LIN {X 0,Y 312.759,Z 483.247,A -85,B 0,C 180,E1 -15907.542,E2 -15907.542} C_VEL
LIN {X 0,Y 310.981,Z 494.774,A -85,B 0,C 180,E1 -15908.976,E2 -15908.976} C_VEL
LIN {X 0,Y 309.46,Z 504.322,A -85,B 0,C 180,E1 -15910.429,E2 -15910.429} C_VEL
LIN {X 0,Y 307.774,Z 514.927,A -85,B 0,C 180,E1 -15912.389,E2 -15912.389} C_VEL
LIN {X 0,Y 306.512,Z 523.604,A -85,B 0,C 180,E1 -15914.368,E2 -15914.368} C_VEL
LIN {X 0,Y 305.528,Z 530.802,A -85,B 0,C 180,E1 -15916.363,E2 -15916.363} C_VEL
LIN {X 0,Y 304.51,Z 537.588,A -85,B 0,C 180,E1 -15918.687,E2 -15918.687} C_VEL
LIN {X 0,Y 304.054,Z 542.26,A -85,B 0,C 180,E1 -15920.689,E2 -15920.689} C_VEL
LIN {X 0,Y 303.769,Z 545.92,A -85,B 0,C 180,E1 -15922.69,E2 -15922.69} C_VEL
LIN {X 0,Y 303.596,Z 548.706,A -85,B 0,C 180,E1 -15924.687,E2 -15924.687} C_VEL
LIN {X 0,Y 303.597,Z 551.095,A -85,B 0,C 180,E1 -15927.346,E2 -15927.346} C_VEL
LIN {X 0,Y 303.603,Z 552.04,A -85,B 0,C 180,E1 -15930,E2 -15930} C_VEL
LIN {X 0,Y 303.597,Z 551.554,A -85,B 0,C 180,E1 -15932.654,E2 -15932.654} C_VEL
LIN {X 0,Y 303.616,Z 549.633,A -85,B 0,C 180,E1 -15935.313,E2 -15935.313} C_VEL
LIN {X 0,Y 303.869,Z 546.198,A -85,B 0,C 180,E1 -15937.977,E2 -15937.977} C_VEL
LIN {X 0,Y 304.429,Z 541.183,A -85,B 0,C 180,E1 -15940.643,E2 -15940.643} C_VEL
LIN {X 0,Y 305.184,Z 536.305,A -85,B 0,C 180,E1 -15942.637,E2 -15942.637} C_VEL
LIN {X 0,Y 306.367,Z 529.293,A -85,B 0,C 180,E1 -15944.93,E2 -15944.93} C_VEL
LIN {X 0,Y 307.58,Z 521.737,A -85,B 0,C 180,E1 -15946.937,E2 -15946.937} C_VEL
LIN {X 0,Y 309.196,Z 512.715,A -85,B 0,C 180,E1 -15948.899,E2 -15948.899} C_VEL
LIN {X 0,Y 311.197,Z 501.739,A -85,B 0,C 180,E1 -15950.836,E2 -15950.836} C_VEL
LIN {X 0,Y 313.164,Z 490.536,A -85,B 0,C 180,E1 -15952.427,E2 -15952.427} C_VEL
LIN {X 0,Y 314.9,Z 478.707,A -85,B 0,C 180,E1 -15953.788,E2 -15953.788} C_VEL
LIN {X 0,Y 316.57,Z 465.924,A -85,B 0,C 180,E1 -15954.948,E2 -15954.948} C_VEL
LIN {X 0,Y 318.089,Z 452.516,A -85,B 0,C 180,E1 -15955.872,E2 -15955.872} C_VEL
LIN {X 0,Y 319.331,Z 438.667,A -85,B 0,C 180,E1 -15956.554,E2 -15956.554} C_VEL
LIN {X 0,Y 320.091,Z 424.187,A -85,B 0,C 180,E1 -15957.014,E2 -15957.014} C_VEL
LIN {X 0,Y 322.808,Z 332.95,A -85,B 0,C 180,E1 -15959.123,E2 -15959.123} C_VEL
LIN {X 0,Y 319.728,Z 313.724,A -85,B 0,C 180,E1 -15959.933,E2 -15959.933} C_VEL
LIN {X 0,Y 313.64,Z 300.106,A -85,B 0,C 180,E1 -15960.977,E2 -15960.977} C_VEL
LIN {X 0,Y 310.945,Z 288.941,A -85,B 0,C 180,E1 -15964.089,E2 -15964.089} C_VEL
LIN {X 0,Y 307.491,Z 276.823,A -85,B 0,C 180,E1 -15967.82,E2 -15967.82} C_VEL
LIN {X 0,Y 305.493,Z 270.13,A -85,B 0,C 180,E1 -15970.101,E2 -15970.101} C_VEL
LIN {X 0,Y 305.488,Z 270.046,A -85,B 0,C 180,E1 -15973.643,E2 -15973.643} C_VEL
LIN {X 0,Y 305.46,Z 270.051,A -85,B 0,C 180,E1 -15977.412,E2 -15977.412} C_VEL
LIN {X 0,Y 305.491,Z 270.058,A -85,B 0,C 180,E1 -15981.6,E2 -15981.6} C_VEL
LIN {X 0,Y 305.458,Z 270.04,A -85,B 0,C 180,E1 -15984.887,E2 -15984.887} C_VEL
LIN {X 0,Y 305.448,Z 270.049,A -85,B 0,C 180,E1 -15988.355,E2 -15988.355} C_VEL
LIN {X 0,Y 305.516,Z 270.026,A -85,B 0,C 180,E1 -15991.114,E2 -15991.114} C_VEL
LIN {X 0,Y 305.567,Z 270.047,A -85,B 0,C 180,E1 -15994.088,E2 -15994.088} C_VEL
LIN {X 0,Y 305.496,Z 270.052,A -85,B 0,C 180,E1 -15998.403,E2 -15998.403} C_VEL
LIN {X 0,Y 305.585,Z 270.044,A -85,B 0,C 180,E1 -16001.218,E2 -16001.218} C_VEL
LIN {X 0,Y 305.644,Z 270.035,A -85,B 0,C 180,E1 -16005.349,E2 -16005.349} C_VEL
LIN {X 0,Y 305.633,Z 270.033,A -85,B 0,C 180,E1 -16009.4,E2 -16009.4} C_VEL
LIN {X 0,Y 305.803,Z 270.006,A -85,B 0,C 180,E1 -16012.074,E2 -16012.074} C_VEL
LIN {X 0,Y 305.683,Z 270.032,A -85,B 0,C 180,E1 -16014.724,E2 -16014.724} C_VEL
LIN {X 0,Y 305.952,Z 269.994,A -85,B 0,C 180,E1 -16018.684,E2 -16018.684} C_VEL
LIN {X 0,Y 305.952,Z 269.991,A -85,B 0,C 180,E1 -16021.317,E2 -16021.317} C_VEL
LIN {X 0,Y 305.848,Z 270.002,A -85,B 0,C 180,E1 -16026.598,E2 -16026.598} C_VEL
LIN {X 0,Y 305.732,Z 270.028,A -85,B 0,C 180,E1 -16029.26,E2 -16029.26} C_VEL
LIN {X 0,Y 305.585,Z 270.044,A -85,B 0,C 180,E1 -16033.297,E2 -16033.297} C_VEL
LIN {X 0,Y 305.59,Z 270.034,A -85,B 0,C 180,E1 -16036.021,E2 -16036.021} C_VEL
LIN {X 0,Y 305.573,Z 270.038,A -85,B 0,C 180,E1 -16039.445,E2 -16039.445} C_VEL
LIN {X 0,Y 305.487,Z 270.053,A -85,B 0,C 180,E1 -16043.042,E2 -16043.042} C_VEL
LIN {X 0,Y 305.544,Z 270.05,A -85,B 0,C 180,E1 -16046.228,E2 -16046.228} C_VEL
LIN {X 0,Y 305.485,Z 270.027,A -85,B 0,C 180,E1 -16049.048,E2 -16049.048} C_VEL
LIN {X 0,Y 305.44,Z 270.064,A -85,B 0,C 180,E1 -16051.953,E2 -16051.953} C_VEL
LIN {X 0,Y 305.461,Z 270.037,A -85,B 0,C 180,E1 -16055.114,E2 -16055.114} C_VEL
LIN {X 0,Y 305.466,Z 270.052,A -85,B 0,C 180,E1 -16058.534,E2 -16058.534} C_VEL
LIN {X 0,Y 305.455,Z 270.06,A -85,B 0,C 180,E1 -16062.587,E2 -16062.587} C_VEL
LIN {X 0,Y 305.426,Z 270.063,A -85,B 0,C 180,E1 -16066.346,E2 -16066.346} C_VEL
LIN {X 0,Y 305.472,Z 270.249,A -85,B 0,C 180,E1 -16067.75,E2 -16067.75} C_VEL
LIN {X 0,Y 308.474,Z 280.592,A -85,B 0,C 180,E1 -16071.315,E2 -16071.315} C_VEL
LIN {X 0,Y 311.024,Z 290.406,A -85,B 0,C 180,E1 -16074.437,E2 -16074.437} C_VEL
LIN {X 0,Y 313.705,Z 302.514,A -85,B 0,C 180,E1 -16078.011,E2 -16078.011} C_VEL
LIN {X 0,Y 314.541,Z 307.647,A -85,B 0,C 180,E1 -16079.448,E2 -16079.448} C_VEL
LIN {X 0,Y 314.073,Z 310.802,A -85,B 0,C 180,E1 -16080.151,E2 -16080.151} C_VEL
LIN {X 0,Y 319.423,Z 338.198,A -85,B 0,C 180,E1 -16081.396,E2 -16081.396} C_VEL
LIN {X 0,Y 321.917,Z 352.925,A -85,B 0,C 180,E1 -16081.99,E2 -16081.99} C_VEL
LIN {X 0,Y 319.923,Z 427.545,A -85,B 0,C 180,E1 -16083.587,E2 -16083.587} C_VEL
LIN {X 0,Y 318.95,Z 440.96,A -85,B 0,C 180,E1 -16084.116,E2 -16084.116} C_VEL
LIN {X 0,Y 317.867,Z 453.812,A -85,B 0,C 180,E1 -16084.898,E2 -16084.898} C_VEL
LIN {X 0,Y 316.415,Z 466.19,A -85,B 0,C 180,E1 -16085.922,E2 -16085.922} C_VEL
LIN {X 0,Y 314.619,Z 477.746,A -85,B 0,C 180,E1 -16087.162,E2 -16087.162} C_VEL
LIN {X 0,Y 312.748,Z 488.241,A -85,B 0,C 180,E1 -16088.583,E2 -16088.583} C_VEL
LIN {X 0,Y 310.959,Z 497.743,A -85,B 0,C 180,E1 -16090.183,E2 -16090.183} C_VEL
LIN {X 0,Y 309.3,Z 505.574,A -85,B 0,C 180,E1 -16091.794,E2 -16091.794} C_VEL
LIN {X 0,Y 307.718,Z 513.396,A -85,B 0,C 180,E1 -16093.776,E2 -16093.776} C_VEL
LIN {X 0,Y 306.336,Z 520.446,A -85,B 0,C 180,E1 -16096.061,E2 -16096.061} C_VEL
LIN {X 0,Y 305.226,Z 525.27,A -85,B 0,C 180,E1 -16098.04,E2 -16098.04} C_VEL
LIN {X 0,Y 304.604,Z 529.037,A -85,B 0,C 180,E1 -16100.035,E2 -16100.035} C_VEL
LIN {X 0,Y 304.12,Z 531.847,A -85,B 0,C 180,E1 -16102.03,E2 -16102.03} C_VEL
LIN {X 0,Y 303.748,Z 534.172,A -85,B 0,C 180,E1 -16104.69,E2 -16104.69} C_VEL
LIN {X 0,Y 303.715,Z 534.785,A -85,B 0,C 180,E1 -16106.019,E2 -16106.019} C_VEL
LIN {X 0,Y 303.602,Z 534.951,A -85,B 0,C 180,E1 -16108.674,E2 -16108.674} C_VEL
LIN {X 0,Y 303.683,Z 533.622,A -85,B 0,C 180,E1 -16111.326,E2 -16111.326} C_VEL
LIN {X 0,Y 304.084,Z 530.811,A -85,B 0,C 180,E1 -16113.976,E2 -16113.976} C_VEL
LIN {X 0,Y 304.569,Z 527.648,A -85,B 0,C 180,E1 -16115.96,E2 -16115.96} C_VEL
LIN {X 0,Y 305.245,Z 523.152,A -85,B 0,C 180,E1 -16118.09,E2 -16118.09} C_VEL
LIN {X 0,Y 306.021,Z 518.261,A -85,B 0,C 180,E1 -16119.918,E2 -16119.918} C_VEL
LIN {X 0,Y 307.428,Z 510.543,A -85,B 0,C 180,E1 -16122.208,E2 -16122.208} C_VEL
LIN {X 0,Y 308.915,Z 502.223,A -85,B 0,C 180,E1 -16124.156,E2 -16124.156} C_VEL
LIN {X 0,Y 310.409,Z 493.744,A -85,B 0,C 180,E1 -16125.765,E2 -16125.765} C_VEL
LIN {X 0,Y 312.086,Z 483.367,A -85,B 0,C 180,E1 -16127.36,E2 -16127.36} C_VEL
LIN {X 0,Y 313.701,Z 471.745,A -85,B 0,C 180,E1 -16128.787,E2 -16128.787} C_VEL
LIN {X 0,Y 315.026,Z 462.036,A -85,B 0,C 180,E1 -16129.72,E2 -16129.72} C_VEL
LIN {X 0,Y 316.343,Z 449.727,A -85,B 0,C 180,E1 -16130.651,E2 -16130.651} C_VEL
LIN {X 0,Y 317.274,Z 436.502,A -85,B 0,C 180,E1 -16131.368,E2 -16131.368} C_VEL
LIN {X 0,Y 317.974,Z 423.135,A -85,B 0,C 180,E1 -16131.816,E2 -16131.816} C_VEL
LIN {X 0,Y 319.599,Z 351.308,A -85,B 0,C 180,E1 -16133.344,E2 -16133.344} C_VEL
LIN {X 0,Y 314.658,Z 321.72,A -85,B 0,C 180,E1 -16134.479,E2 -16134.479} C_VEL
LIN {X 0,Y 312.643,Z 310.757,A -85,B 0,C 180,E1 -16134.972,E2 -16134.972} C_VEL
LIN {X 0,Y 313.465,Z 303.711,A -85,B 0,C 180,E1 -16136.641,E2 -16136.641} C_VEL
LIN {X 0,Y 311.277,Z 292.524,A -85,B 0,C 180,E1 -16139.782,E2 -16139.782} C_VEL
LIN {X 0,Y 308.2,Z 280.123,A -85,B 0,C 180,E1 -16143.526,E2 -16143.526} C_VEL
LIN {X 0,Y 305.574,Z 270.458,A -85,B 0,C 180,E1 -16146.661,E2 -16146.661} C_VEL
LIN {X 0,Y 305.318,Z 270.1,A -85,B 0,C 180,E1 -16146.986,E2 -16146.986} C_VEL
LIN {X 0,Y 302.785,Z 270.39,A -85,B 0,C 180,E1 -16148.741,E2 -16148.741} C_VEL
LIN {X 0,Y 299.323,Z 271.015,A -85,B 0,C 180,E1 -16150.95,E2 -16150.95} C_VEL
LIN {X 0,Y 298.422,Z 270.949,A -85,B 0,C 180,E1 -16152.109,E2 -16152.109} C_VEL
LIN {X 0,Y 298.364,Z 270.938,A -85,B 0,C 180,E1 -16152.501,E2 -16152.501} C_VEL
LIN {X 0,Y 298.402,Z 270.937,A -85,B 0,C 180,E1 -16156.92,E2 -16156.92} C_VEL
LIN {X 0,Y 298.413,Z 270.917,A -85,B 0,C 180,E1 -16161.003,E2 -16161.003} C_VEL
LIN {X 0,Y 298.43,Z 270.933,A -85,B 0,C 180,E1 -16163.931,E2 -16163.931} C_VEL
LIN {X 0,Y 298.393,Z 270.924,A -85,B 0,C 180,E1 -16167.982,E2 -16167.982} C_VEL
LIN {X 0,Y 298.467,Z 270.922,A -85,B 0,C 180,E1 -16171.904,E2 -16171.904} C_VEL
LIN {X 0,Y 298.482,Z 270.923,A -85,B 0,C 180,E1 -16174.923,E2 -16174.923} C_VEL
LIN {X 0,Y 298.446,Z 270.927,A -85,B 0,C 180,E1 -16179.314,E2 -16179.314} C_VEL
LIN {X 0,Y 298.534,Z 270.922,A -85,B 0,C 180,E1 -16182.179,E2 -16182.179} C_VEL
LIN {X 0,Y 298.589,Z 270.905,A -85,B 0,C 180,E1 -16184.994,E2 -16184.994} C_VEL
LIN {X 0,Y 298.587,Z 270.908,A -85,B 0,C 180,E1 -16189.146,E2 -16189.146} C_VEL
LIN {X 0,Y 298.736,Z 270.895,A -85,B 0,C 180,E1 -16191.885,E2 -16191.885} C_VEL
LIN {X 0,Y 298.652,Z 270.897,A -85,B 0,C 180,E1 -16194.598,E2 -16194.598} C_VEL
LIN {X 0,Y 298.918,Z 270.874,A -85,B 0,C 180,E1 -16198.652,E2 -16198.652} C_VEL
LIN {X 0,Y 298.918,Z 270.865,A -85,B 0,C 180,E1 -16201.347,E2 -16201.347} C_VEL
LIN {X 0,Y 298.792,Z 270.881,A -85,B 0,C 180,E1 -16206.754,E2 -16206.754} C_VEL
LIN {X 0,Y 298.675,Z 270.903,A -85,B 0,C 180,E1 -16209.48,E2 -16209.48} C_VEL
LIN {X 0,Y 298.546,Z 270.922,A -85,B 0,C 180,E1 -16213.615,E2 -16213.615} C_VEL
LIN {X 0,Y 298.543,Z 270.912,A -85,B 0,C 180,E1 -16216.409,E2 -16216.409} C_VEL
LIN {X 0,Y 298.506,Z 270.921,A -85,B 0,C 180,E1 -16219.655,E2 -16219.655} C_VEL
LIN {X 0,Y 298.452,Z 270.932,A -85,B 0,C 180,E1 -16223.598,E2 -16223.598} C_VEL
LIN {X 0,Y 298.485,Z 270.93,A -85,B 0,C 180,E1 -16226.574,E2 -16226.574} C_VEL
LIN {X 0,Y 298.416,Z 270.908,A -85,B 0,C 180,E1 -16229.641,E2 -16229.641} C_VEL
LIN {X 0,Y 298.391,Z 270.936,A -85,B 0,C 180,E1 -16232.8,E2 -16232.8} C_VEL
LIN {X 0,Y 298.442,Z 270.909,A -85,B 0,C 180,E1 -16236.808,E2 -16236.808} C_VEL
LIN {X 0,Y 298.383,Z 270.93,A -85,B 0,C 180,E1 -16241.088,E2 -16241.088} C_VEL
LIN {X 0,Y 298.385,Z 270.935,A -85,B 0,C 180,E1 -16245.042,E2 -16245.042} C_VEL
LIN {X 0,Y 298.384,Z 270.886,A -85,B 0,C 180,E1 -16248.913,E2 -16248.913} C_VEL
LIN {X 0,Y 298.422,Z 271.119,A -85,B 0,C 180,E1 -16250.769,E2 -16250.769} C_VEL
LIN {X 0,Y 301.752,Z 282.523,A -85,B 0,C 180,E1 -16254.391,E2 -16254.391} C_VEL
LIN {X 0,Y 304.525,Z 293.397,A -85,B 0,C 180,E1 -16257.58,E2 -16257.58} C_VEL
LIN {X 0,Y 306.122,Z 300.383,A -85,B 0,C 180,E1 -16259.437,E2 -16259.437} C_VEL
LIN {X 0,Y 311.319,Z 312.764,A -85,B 0,C 180,E1 -16260.308,E2 -16260.308} C_VEL
LIN {X 0,Y 314.225,Z 333.621,A -85,B 0,C 180,E1 -16261.127,E2 -16261.127} C_VEL
LIN {X 0,Y 311.299,Z 430.528,A -85,B 0,C 180,E1 -16263.43,E2 -16263.43} C_VEL
LIN {X 0,Y 310.325,Z 445.033,A -85,B 0,C 180,E1 -16264.019,E2 -16264.019} C_VEL
LIN {X 0,Y 309.172,Z 457.738,A -85,B 0,C 180,E1 -16264.773,E2 -16264.773} C_VEL
LIN {X 0,Y 307.655,Z 471.105,A -85,B 0,C 180,E1 -16265.838,E2 -16265.838} C_VEL
LIN {X 0,Y 306.161,Z 482.751,A -85,B 0,C 180,E1 -16267.031,E2 -16267.031} C_VEL
LIN {X 0,Y 304.322,Z 494.343,A -85,B 0,C 180,E1 -16268.493,E2 -16268.493} C_VEL
LIN {X 0,Y 302.685,Z 503.937,A -85,B 0,C 180,E1 -16269.973,E2 -16269.973} C_VEL
LIN {X 0,Y 300.971,Z 514.584,A -85,B 0,C 180,E1 -16271.977,E2 -16271.977} C_VEL
LIN {X 0,Y 299.496,Z 523.967,A -85,B 0,C 180,E1 -16274.176,E2 -16274.176} C_VEL
LIN {X 0,Y 298.548,Z 530.514,A -85,B 0,C 180,E1 -16276.038,E2 -16276.038} C_VEL
LIN {X 0,Y 297.511,Z 537.328,A -85,B 0,C 180,E1 -16278.417,E2 -16278.417} C_VEL
LIN {X 0,Y 297.004,Z 542.007,A -85,B 0,C 180,E1 -16280.466,E2 -16280.466} C_VEL
LIN {X 0,Y 296.69,Z 545.683,A -85,B 0,C 180,E1 -16282.514,E2 -16282.514} C_VEL
LIN {X 0,Y 296.511,Z 548.482,A -85,B 0,C 180,E1 -16284.56,E2 -16284.56} C_VEL
LIN {X 0,Y 296.522,Z 550.884,A -85,B 0,C 180,E1 -16287.283,E2 -16287.283} C_VEL
LIN {X 0,Y 296.518,Z 551.839,A -85,B 0,C 180,E1 -16290,E2 -16290} C_VEL
LIN {X 0,Y 296.522,Z 551.362,A -85,B 0,C 180,E1 -16292.717,E2 -16292.717} C_VEL
LIN {X 0,Y 296.545,Z 549.383,A -85,B 0,C 180,E1 -16295.509,E2 -16295.509} C_VEL
LIN {X 0,Y 296.814,Z 546.027,A -85,B 0,C 180,E1 -16298.168,E2 -16298.168} C_VEL
LIN {X 0,Y 297.388,Z 541.019,A -85,B 0,C 180,E1 -16300.898,E2 -16300.898} C_VEL
LIN {X 0,Y 298.229,Z 536.149,A -85,B 0,C 180,E1 -16302.937,E2 -16302.937} C_VEL
LIN {X 0,Y 299.259,Z 530.192,A -85,B 0,C 180,E1 -16304.971,E2 -16304.971} C_VEL
LIN {X 0,Y 300.527,Z 522.967,A -85,B 0,C 180,E1 -16306.997,E2 -16306.997} C_VEL
LIN {X 0,Y 302.149,Z 514.222,A -85,B 0,C 180,E1 -16309.004,E2 -16309.004} C_VEL
LIN {X 0,Y 304.15,Z 503.571,A -85,B 0,C 180,E1 -16310.987,E2 -16310.987} C_VEL
LIN {X 0,Y 306.156,Z 492.777,A -85,B 0,C 180,E1 -16312.613,E2 -16312.613} C_VEL
LIN {X 0,Y 308.1,Z 480.527,A -85,B 0,C 180,E1 -16314.112,E2 -16314.112} C_VEL
LIN {X 0,Y 309.917,Z 467.747,A -85,B 0,C 180,E1 -16315.342,E2 -16315.342} C_VEL
LIN {X 0,Y 311.443,Z 454.922,A -85,B 0,C 180,E1 -16316.286,E2 -16316.286} C_VEL
LIN {X 0,Y 312.757,Z 441.147,A -85,B 0,C 180,E1 -16317.022,E2 -16317.022} C_VEL
LIN {X 0,Y 313.656,Z 426.797,A -85,B 0,C 180,E1 -16317.525,E2 -16317.525} C_VEL
LIN {X 0,Y 316.583,Z 334.1,A -85,B 0,C 180,E1 -16319.709,E2 -16319.709} C_VEL
LIN {X 0,Y 313.725,Z 316.254,A -85,B 0,C 180,E1 -16320.485,E2 -16320.485} C_VEL
LIN {X 0,Y 306.546,Z 300.388,A -85,B 0,C 180,E1 -16321.739,E2 -16321.739} C_VEL
LIN {X 0,Y 303.827,Z 289.344,A -85,B 0,C 180,E1 -16324.924,E2 -16324.924} C_VEL
LIN {X 0,Y 300.648,Z 278.286,A -85,B 0,C 180,E1 -16328.456,E2 -16328.456} C_VEL
LIN {X 0,Y 298.452,Z 271.029,A -85,B 0,C 180,E1 -16330.983,E2 -16330.983} C_VEL
LIN {X 0,Y 298.456,Z 270.928,A -85,B 0,C 180,E1 -16333.115,E2 -16333.115} C_VEL
LIN {X 0,Y 298.429,Z 270.935,A -85,B 0,C 180,E1 -16336.926,E2 -16336.926} C_VEL
LIN {X 0,Y 298.411,Z 270.94,A -85,B 0,C 180,E1 -16341.003,E2 -16341.003} C_VEL
LIN {X 0,Y 298.416,Z 270.912,A -85,B 0,C 180,E1 -16343.93,E2 -16343.93} C_VEL
LIN {X 0,Y 298.391,Z 270.933,A -85,B 0,C 180,E1 -16347.983,E2 -16347.983} C_VEL
LIN {X 0,Y 298.459,Z 270.915,A -85,B 0,C 180,E1 -16351.904,E2 -16351.904} C_VEL
LIN {X 0,Y 298.481,Z 270.924,A -85,B 0,C 180,E1 -16354.924,E2 -16354.924} C_VEL
LIN {X 0,Y 298.445,Z 270.925,A -85,B 0,C 180,E1 -16359.315,E2 -16359.315} C_VEL
LIN {X 0,Y 298.533,Z 270.921,A -85,B 0,C 180,E1 -16362.179,E2 -16362.179} C_VEL
LIN {X 0,Y 298.589,Z 270.912,A -85,B 0,C 180,E1 -16364.995,E2 -16364.995} C_VEL
LIN {X 0,Y 298.588,Z 270.909,A -85,B 0,C 180,E1 -16369.147,E2 -16369.147} C_VEL
LIN {X 0,Y 298.75,Z 270.886,A -85,B 0,C 180,E1 -16371.886,E2 -16371.886} C_VEL
LIN {X 0,Y 298.654,Z 270.907,A -85,B 0,C 180,E1 -16374.599,E2 -16374.599} C_VEL
LIN {X 0,Y 298.919,Z 270.87,A -85,B 0,C 180,E1 -16378.653,E2 -16378.653} C_VEL
LIN {X 0,Y 298.919,Z 270.867,A -85,B 0,C 180,E1 -16381.348,E2 -16381.348} C_VEL
LIN {X 0,Y 298.793,Z 270.879,A -85,B 0,C 180,E1 -16386.754,E2 -16386.754} C_VEL
LIN {X 0,Y 298.677,Z 270.906,A -85,B 0,C 180,E1 -16389.481,E2 -16389.481} C_VEL
LIN {X 0,Y 298.548,Z 270.922,A -85,B 0,C 180,E1 -16393.616,E2 -16393.616} C_VEL
LIN {X 0,Y 298.545,Z 270.913,A -85,B 0,C 180,E1 -16396.409,E2 -16396.409} C_VEL
LIN {X 0,Y 298.508,Z 270.917,A -85,B 0,C 180,E1 -16399.655,E2 -16399.655} C_VEL
LIN {X 0,Y 298.455,Z 270.925,A -85,B 0,C 180,E1 -16403.599,E2 -16403.599} C_VEL
LIN {X 0,Y 298.487,Z 270.925,A -85,B 0,C 180,E1 -16406.575,E2 -16406.575} C_VEL
LIN {X 0,Y 298.414,Z 270.909,A -85,B 0,C 180,E1 -16409.642,E2 -16409.642} C_VEL
LIN {X 0,Y 298.393,Z 270.939,A -85,B 0,C 180,E1 -16412.801,E2 -16412.801} C_VEL
LIN {X 0,Y 298.463,Z 270.925,A -85,B 0,C 180,E1 -16416.813,E2 -16416.813} C_VEL
LIN {X 0,Y 298.386,Z 270.928,A -85,B 0,C 180,E1 -16421.088,E2 -16421.088} C_VEL
LIN {X 0,Y 298.399,Z 270.931,A -85,B 0,C 180,E1 -16423.104,E2 -16423.104} C_VEL
LIN {X 0,Y 298.422,Z 271.135,A -85,B 0,C 180,E1 -16426.847,E2 -16426.847} C_VEL
LIN {X 0,Y 301.273,Z 280.862,A -85,B 0,C 180,E1 -16430.338,E2 -16430.338} C_VEL
LIN {X 0,Y 304.224,Z 291.819,A -85,B 0,C 180,E1 -16433.955,E2 -16433.955} C_VEL
LIN {X 0,Y 307.023,Z 304.814,A -85,B 0,C 180,E1 -16437.884,E2 -16437.884} C_VEL
LIN {X 0,Y 307.738,Z 309.703,A -85,B 0,C 180,E1 -16439.271,E2 -16439.271} C_VEL
LIN {X 0,Y 307.638,Z 310.773,A -85,B 0,C 180,E1 -16439.46,E2 -16439.46} C_VEL
LIN {X 0,Y 312.585,Z 335.948,A -85,B 0,C 180,E1 -16440.646,E2 -16440.646} C_VEL
LIN {X 0,Y 315.647,Z 354.231,A -85,B 0,C 180,E1 -16441.408,E2 -16441.408} C_VEL
LIN {X 0,Y 313.648,Z 426.468,A -85,B 0,C 180,E1 -16442.971,E2 -16442.971} C_VEL
LIN {X 0,Y 312.739,Z 439.521,A -85,B 0,C 180,E1 -16443.472,E2 -16443.472} C_VEL
LIN {X 0,Y 311.534,Z 452.773,A -85,B 0,C 180,E1 -16444.262,E2 -16444.262} C_VEL
LIN {X 0,Y 310.122,Z 464.797,A -85,B 0,C 180,E1 -16445.245,E2 -16445.245} C_VEL
LIN {X 0,Y 308.33,Z 476.561,A -85,B 0,C 180,E1 -16446.492,E2 -16446.492} C_VEL
LIN {X 0,Y 306.35,Z 487.287,A -85,B 0,C 180,E1 -16447.935,E2 -16447.935} C_VEL
LIN {X 0,Y 304.601,Z 496.096,A -85,B 0,C 180,E1 -16449.399,E2 -16449.399} C_VEL
LIN {X 0,Y 302.531,Z 505.695,A -85,B 0,C 180,E1 -16451.372,E2 -16451.372} C_VEL
LIN {X 0,Y 300.992,Z 512.839,A -85,B 0,C 180,E1 -16453.204,E2 -16453.204} C_VEL
LIN {X 0,Y 299.858,Z 518.72,A -85,B 0,C 180,E1 -16455.06,E2 -16455.06} C_VEL
LIN {X 0,Y 298.593,Z 523.933,A -85,B 0,C 180,E1 -16457.079,E2 -16457.079} C_VEL
LIN {X 0,Y 297.769,Z 528.04,A -85,B 0,C 180,E1 -16459.116,E2 -16459.116} C_VEL
LIN {X 0,Y 297.412,Z 530.234,A -85,B 0,C 180,E1 -16460.479,E2 -16460.479} C_VEL
LIN {X 0,Y 297.07,Z 532.019,A -85,B 0,C 180,E1 -16461.84,E2 -16461.84} C_VEL
LIN {X 0,Y 296.672,Z 534.356,A -85,B 0,C 180,E1 -16464.563,E2 -16464.563} C_VEL
LIN {X 0,Y 296.574,Z 535.24,A -85,B 0,C 180,E1 -16467.283,E2 -16467.283} C_VEL
LIN {X 0,Y 296.528,Z 534.688,A -85,B 0,C 180,E1 -16470,E2 -16470} C_VEL
LIN {X 0,Y 296.762,Z 532.631,A -85,B 0,C 180,E1 -16472.715,E2 -16472.715} C_VEL
LIN {X 0,Y 297.355,Z 529.071,A -85,B 0,C 180,E1 -16475.425,E2 -16475.425} C_VEL
LIN {X 0,Y 297.897,Z 525.39,A -85,B 0,C 180,E1 -16477.398,E2 -16477.398} C_VEL
LIN {X 0,Y 298.696,Z 520.427,A -85,B 0,C 180,E1 -16479.48,E2 -16479.48} C_VEL
LIN {X 0,Y 299.801,Z 514.388,A -85,B 0,C 180,E1 -16481.493,E2 -16481.493} C_VEL
LIN {X 0,Y 301.287,Z 506.941,A -85,B 0,C 180,E1 -16483.489,E2 -16483.489} C_VEL
LIN {X 0,Y 302.676,Z 499.386,A -85,B 0,C 180,E1 -16485.142,E2 -16485.142} C_VEL
LIN {X 0,Y 304.386,Z 489.266,A -85,B 0,C 180,E1 -16486.947,E2 -16486.947} C_VEL
LIN {X 0,Y 306.108,Z 479.014,A -85,B 0,C 180,E1 -16488.402,E2 -16488.402} C_VEL
LIN {X 0,Y 307.518,Z 469.278,A -85,B 0,C 180,E1 -16489.526,E2 -16489.526} C_VEL
LIN {X 0,Y 309.054,Z 457.012,A -85,B 0,C 180,E1 -16490.638,E2 -16490.638} C_VEL
LIN {X 0,Y 310.233,Z 444.565,A -85,B 0,C 180,E1 -16491.486,E2 -16491.486} C_VEL
LIN {X 0,Y 311.151,Z 431.625,A -85,B 0,C 180,E1 -16492.09,E2 -16492.09} C_VEL
LIN {X 0,Y 311.7,Z 416.204,A -85,B 0,C 180,E1 -16492.508,E2 -16492.508} C_VEL
LIN {X 0,Y 313.152,Z 351.889,A -85,B 0,C 180,E1 -16493.901,E2 -16493.901} C_VEL
LIN {X 0,Y 308.103,Z 321.447,A -85,B 0,C 180,E1 -16495.108,E2 -16495.108} C_VEL
LIN {X 0,Y 306.091,Z 310.752,A -85,B 0,C 180,E1 -16495.599,E2 -16495.599} C_VEL
LIN {X 0,Y 306.673,Z 305.551,A -85,B 0,C 180,E1 -16496.829,E2 -16496.829} C_VEL
LIN {X 0,Y 304.742,Z 295.455,A -85,B 0,C 180,E1 -16499.723,E2 -16499.723} C_VEL
LIN {X 0,Y 301.852,Z 283.472,A -85,B 0,C 180,E1 -16503.4,E2 -16503.4} C_VEL
LIN {X 0,Y 298.928,Z 272.785,A -85,B 0,C 180,E1 -16506.93,E2 -16506.93} C_VEL
LIN {X 0,Y 298.458,Z 270.999,A -85,B 0,C 180,E1 -16507.618,E2 -16507.618} C_VEL
LIN {X 0,Y 298.384,Z 270.929,A -85,B 0,C 180,E1 -16511.261,E2 -16511.261} C_VEL
LIN {X 0,Y 298.364,Z 270.938,A -85,B 0,C 180,E1 -16512.501,E2 -16512.501} C_VEL
LIN {X 0,Y 297.738,Z 271.029,A -85,B 0,C 180,E1 -16513.628,E2 -16513.628} C_VEL
LIN {X 0,Y 294.904,Z 271.392,A -85,B 0,C 180,E1 -16515.463,E2 -16515.463} C_VEL
LIN {X 0,Y 292.47,Z 271.689,A -85,B 0,C 180,E1 -16516.953,E2 -16516.953} C_VEL
LIN {X 0,Y 291.413,Z 271.808,A -85,B 0,C 180,E1 -16518.106,E2 -16518.106} C_VEL
LIN {X 0,Y 291.322,Z 271.811,A -85,B 0,C 180,E1 -16518.498,E2 -16518.498} C_VEL
LIN {X 0,Y 291.363,Z 271.796,A -85,B 0,C 180,E1 -16521.159,E2 -16521.159} C_VEL
LIN {X 0,Y 291.383,Z 271.797,A -85,B 0,C 180,E1 -16524.628,E2 -16524.628} C_VEL
LIN {X 0,Y 291.37,Z 271.797,A -85,B 0,C 180,E1 -16527.95,E2 -16527.95} C_VEL
LIN {X 0,Y 291.382,Z 271.807,A -85,B 0,C 180,E1 -16531.158,E2 -16531.158} C_VEL
LIN {X 0,Y 291.418,Z 271.81,A -85,B 0,C 180,E1 -16534.271,E2 -16534.271} C_VEL
LIN {X 0,Y 291.377,Z 271.814,A -85,B 0,C 180,E1 -16537.299,E2 -16537.299} C_VEL
LIN {X 0,Y 291.455,Z 271.794,A -85,B 0,C 180,E1 -16540.269,E2 -16540.269} C_VEL
LIN {X 0,Y 291.536,Z 271.784,A -85,B 0,C 180,E1 -16544.634,E2 -16544.634} C_VEL
LIN {X 0,Y 291.531,Z 271.788,A -85,B 0,C 180,E1 -16548.88,E2 -16548.88} C_VEL
LIN {X 0,Y 291.683,Z 271.773,A -85,B 0,C 180,E1 -16551.687,E2 -16551.687} C_VEL
LIN {X 0,Y 291.622,Z 271.773,A -85,B 0,C 180,E1 -16554.468,E2 -16554.468} C_VEL
LIN {X 0,Y 291.884,Z 271.75,A -85,B 0,C 180,E1 -16558.62,E2 -16558.62} C_VEL
LIN {X 0,Y 291.884,Z 271.741,A -85,B 0,C 180,E1 -16561.379,E2 -16561.379} C_VEL
LIN {X 0,Y 291.741,Z 271.761,A -85,B 0,C 180,E1 -16566.918,E2 -16566.918} C_VEL
LIN {X 0,Y 291.624,Z 271.78,A -85,B 0,C 180,E1 -16569.712,E2 -16569.712} C_VEL
LIN {X 0,Y 291.516,Z 271.799,A -85,B 0,C 180,E1 -16573.95,E2 -16573.95} C_VEL
LIN {X 0,Y 291.482,Z 271.795,A -85,B 0,C 180,E1 -16576.818,E2 -16576.818} C_VEL
LIN {X 0,Y 291.446,Z 271.798,A -85,B 0,C 180,E1 -16579.875,E2 -16579.875} C_VEL
LIN {X 0,Y 291.395,Z 271.805,A -85,B 0,C 180,E1 -16584.205,E2 -16584.205} C_VEL
LIN {X 0,Y 291.418,Z 271.81,A -85,B 0,C 180,E1 -16587.272,E2 -16587.272} C_VEL
LIN {X 0,Y 291.332,Z 271.787,A -85,B 0,C 180,E1 -16590.437,E2 -16590.437} C_VEL
LIN {X 0,Y 291.34,Z 271.822,A -85,B 0,C 180,E1 -16593.699,E2 -16593.699} C_VEL
LIN {X 0,Y 291.372,Z 271.791,A -85,B 0,C 180,E1 -16597.254,E2 -16597.254} C_VEL
LIN {X 0,Y 291.329,Z 271.815,A -85,B 0,C 180,E1 -16600.643,E2 -16600.643} C_VEL
LIN {X 0,Y 291.312,Z 271.824,A -85,B 0,C 180,E1 -16604.397,E2 -16604.397} C_VEL
LIN {X 0,Y 291.323,Z 271.761,A -85,B 0,C 180,E1 -16608.405,E2 -16608.405} C_VEL
LIN {X 0,Y 291.356,Z 272,A -85,B 0,C 180,E1 -16609.918,E2 -16609.918} C_VEL
LIN {X 0,Y 294.772,Z 283.523,A -85,B 0,C 180,E1 -16613.724,E2 -16613.724} C_VEL
LIN {X 0,Y 297.888,Z 295.768,A -85,B 0,C 180,E1 -16617.42,E2 -16617.42} C_VEL
LIN {X 0,Y 298.984,Z 300.489,A -85,B 0,C 180,E1 -16618.698,E2 -16618.698} C_VEL
LIN {X 0,Y 305.18,Z 314.984,A -85,B 0,C 180,E1 -16619.767,E2 -16619.767} C_VEL
LIN {X 0,Y 307.879,Z 334.862,A -85,B 0,C 180,E1 -16620.566,E2 -16620.566} C_VEL
LIN {X 0,Y 304.805,Z 431.437,A -85,B 0,C 180,E1 -16622.911,E2 -16622.911} C_VEL
LIN {X 0,Y 303.785,Z 445.606,A -85,B 0,C 180,E1 -16623.509,E2 -16623.509} C_VEL
LIN {X 0,Y 302.616,Z 458.149,A -85,B 0,C 180,E1 -16624.279,E2 -16624.279} C_VEL
LIN {X 0,Y 301.108,Z 470.821,A -85,B 0,C 180,E1 -16625.309,E2 -16625.309} C_VEL
LIN {X 0,Y 299.594,Z 482.256,A -85,B 0,C 180,E1 -16626.498,E2 -16626.498} C_VEL
LIN {X 0,Y 297.684,Z 493.913,A -85,B 0,C 180,E1 -16627.989,E2 -16627.989} C_VEL
LIN {X 0,Y 295.968,Z 503.554,A -85,B 0,C 180,E1 -16629.498,E2 -16629.498} C_VEL
LIN {X 0,Y 294.161,Z 514.238,A -85,B 0,C 180,E1 -16631.545,E2 -16631.545} C_VEL
LIN {X 0,Y 292.656,Z 523.497,A -85,B 0,C 180,E1 -16633.749,E2 -16633.749} C_VEL
LIN {X 0,Y 291.585,Z 530.224,A -85,B 0,C 180,E1 -16635.697,E2 -16635.697} C_VEL
LIN {X 0,Y 290.527,Z 537.068,A -85,B 0,C 180,E1 -16638.135,E2 -16638.135} C_VEL
LIN {X 0,Y 289.971,Z 541.754,A -85,B 0,C 180,E1 -16640.232,E2 -16640.232} C_VEL
LIN {X 0,Y 289.638,Z 545.446,A -85,B 0,C 180,E1 -16642.331,E2 -16642.331} C_VEL
LIN {X 0,Y 289.409,Z 548.496,A -85,B 0,C 180,E1 -16644.648,E2 -16644.648} C_VEL
LIN {X 0,Y 289.425,Z 550.672,A -85,B 0,C 180,E1 -16647.216,E2 -16647.216} C_VEL
LIN {X 0,Y 289.435,Z 551.638,A -85,B 0,C 180,E1 -16650,E2 -16650} C_VEL
LIN {X 0,Y 289.425,Z 551.171,A -85,B 0,C 180,E1 -16652.784,E2 -16652.784} C_VEL
LIN {X 0,Y 289.475,Z 549.271,A -85,B 0,C 180,E1 -16655.573,E2 -16655.573} C_VEL
LIN {X 0,Y 289.751,Z 545.856,A -85,B 0,C 180,E1 -16658.368,E2 -16658.368} C_VEL
LIN {X 0,Y 290.357,Z 540.855,A -85,B 0,C 180,E1 -16661.165,E2 -16661.165} C_VEL
LIN {X 0,Y 291.256,Z 535.992,A -85,B 0,C 180,E1 -16663.252,E2 -16663.252} C_VEL
LIN {X 0,Y 292.59,Z 528.937,A -85,B 0,C 180,E1 -16665.667,E2 -16665.667} C_VEL
LIN {X 0,Y 294.19,Z 520.07,A -85,B 0,C 180,E1 -16668.093,E2 -16668.093} C_VEL
LIN {X 0,Y 296.074,Z 510.785,A -85,B 0,C 180,E1 -16670.132,E2 -16670.132} C_VEL
LIN {X 0,Y 298.083,Z 500.452,A -85,B 0,C 180,E1 -16671.98,E2 -16671.98} C_VEL
LIN {X 0,Y 300.042,Z 490.259,A -85,B 0,C 180,E1 -16673.465,E2 -16673.465} C_VEL
LIN {X 0,Y 302.026,Z 477.761,A -85,B 0,C 180,E1 -16674.945,E2 -16674.945} C_VEL
LIN {X 0,Y 303.726,Z 465.615,A -85,B 0,C 180,E1 -16676.081,E2 -16676.081} C_VEL
LIN {X 0,Y 305.387,Z 452.166,A -85,B 0,C 180,E1 -16677.033,E2 -16677.033} C_VEL
LIN {X 0,Y 306.707,Z 438.23,A -85,B 0,C 180,E1 -16677.739,E2 -16677.739} C_VEL
LIN {X 0,Y 307.45,Z 425.02,A -85,B 0,C 180,E1 -16678.175,E2 -16678.175} C_VEL
LIN {X 0,Y 310.352,Z 335.004,A -85,B 0,C 180,E1 -16680.331,E2 -16680.331} C_VEL
LIN {X 0,Y 307.879,Z 319.036,A -85,B 0,C 180,E1 -16681.037,E2 -16681.037} C_VEL
LIN {X 0,Y 299.844,Z 301.564,A -85,B 0,C 180,E1 -16682.457,E2 -16682.457} C_VEL
LIN {X 0,Y 299.313,Z 300.205,A -85,B 0,C 180,E1 -16682.638,E2 -16682.638} C_VEL
LIN {X 0,Y 296.675,Z 289.723,A -85,B 0,C 180,E1 -16685.82,E2 -16685.82} C_VEL
LIN {X 0,Y 293.625,Z 279.083,A -85,B 0,C 180,E1 -16689.354,E2 -16689.354} C_VEL
LIN {X 0,Y 291.404,Z 271.883,A -85,B 0,C 180,E1 -16691.983,E2 -16691.983} C_VEL
LIN {X 0,Y 291.345,Z 271.82,A -85,B 0,C 180,E1 -16696.358,E2 -16696.358} C_VEL
LIN {X 0,Y 291.383,Z 271.809,A -85,B 0,C 180,E1 -16700.517,E2 -16700.517} C_VEL
LIN {X 0,Y 291.41,Z 271.79,A -85,B 0,C 180,E1 -16702.92,E2 -16702.92} C_VEL
LIN {X 0,Y 291.341,Z 271.816,A -85,B 0,C 180,E1 -16706.301,E2 -16706.301} C_VEL
LIN {X 0,Y 291.383,Z 271.78,A -85,B 0,C 180,E1 -16710.26,E2 -16710.26} C_VEL
LIN {X 0,Y 291.413,Z 271.808,A -85,B 0,C 180,E1 -16714.272,E2 -16714.272} C_VEL
LIN {X 0,Y 291.377,Z 271.815,A -85,B 0,C 180,E1 -16717.3,E2 -16717.3} C_VEL
LIN {X 0,Y 291.454,Z 271.798,A -85,B 0,C 180,E1 -16720.27,E2 -16720.27} C_VEL
LIN {X 0,Y 291.551,Z 271.786,A -85,B 0,C 180,E1 -16724.624,E2 -16724.624} C_VEL
LIN {X 0,Y 291.532,Z 271.786,A -85,B 0,C 180,E1 -16728.881,E2 -16728.881} C_VEL
LIN {X 0,Y 291.701,Z 271.766,A -85,B 0,C 180,E1 -16731.689,E2 -16731.689} C_VEL
LIN {X 0,Y 291.624,Z 271.783,A -85,B 0,C 180,E1 -16734.469,E2 -16734.469} C_VEL
LIN {X 0,Y 291.885,Z 271.746,A -85,B 0,C 180,E1 -16738.621,E2 -16738.621} C_VEL
LIN {X 0,Y 291.885,Z 271.742,A -85,B 0,C 180,E1 -16741.38,E2 -16741.38} C_VEL
LIN {X 0,Y 291.742,Z 271.757,A -85,B 0,C 180,E1 -16746.919,E2 -16746.919} C_VEL
LIN {X 0,Y 291.626,Z 271.782,A -85,B 0,C 180,E1 -16749.713,E2 -16749.713} C_VEL
LIN {X 0,Y 291.518,Z 271.796,A -85,B 0,C 180,E1 -16753.951,E2 -16753.951} C_VEL
LIN {X 0,Y 291.484,Z 271.795,A -85,B 0,C 180,E1 -16756.819,E2 -16756.819} C_VEL
LIN {X 0,Y 291.448,Z 271.796,A -85,B 0,C 180,E1 -16759.876,E2 -16759.876} C_VEL
LIN {X 0,Y 291.398,Z 271.805,A -85,B 0,C 180,E1 -16764.206,E2 -16764.206} C_VEL
LIN {X 0,Y 291.419,Z 271.795,A -85,B 0,C 180,E1 -16767.273,E2 -16767.273} C_VEL
LIN {X 0,Y 291.332,Z 271.799,A -85,B 0,C 180,E1 -16770.438,E2 -16770.438} C_VEL
LIN {X 0,Y 291.343,Z 271.804,A -85,B 0,C 180,E1 -16773.699,E2 -16773.699} C_VEL
LIN {X 0,Y 291.393,Z 271.811,A -85,B 0,C 180,E1 -16777.26,E2 -16777.26} C_VEL
LIN {X 0,Y 291.333,Z 271.802,A -85,B 0,C 180,E1 -16780.643,E2 -16780.643} C_VEL
LIN {X 0,Y 291.29,Z 271.811,A -85,B 0,C 180,E1 -16784.403,E2 -16784.403} C_VEL
LIN {X 0,Y 291.387,Z 272.087,A -85,B 0,C 180,E1 -16785.912,E2 -16785.912} C_VEL
LIN {X 0,Y 294.587,Z 282.8,A -85,B 0,C 180,E1 -16789.899,E2 -16789.899} C_VEL
LIN {X 0,Y 297.403,Z 293.292,A -85,B 0,C 180,E1 -16793.463,E2 -16793.463} C_VEL
LIN {X 0,Y 299.822,Z 304.543,A -85,B 0,C 180,E1 -16796.976,E2 -16796.976} C_VEL
LIN {X 0,Y 301.005,Z 310.393,A -85,B 0,C 180,E1 -16798.675,E2 -16798.675} C_VEL
LIN {X 0,Y 302.159,Z 315.224,A -85,B 0,C 180,E1 -16798.977,E2 -16798.977} C_VEL
LIN {X 0,Y 307.494,Z 343.175,A -85,B 0,C 180,E1 -16800.288,E2 -16800.288} C_VEL
LIN {X 0,Y 309.411,Z 355.255,A -85,B 0,C 180,E1 -16800.795,E2 -16800.795} C_VEL
LIN {X 0,Y 307.46,Z 423.543,A -85,B 0,C 180,E1 -16802.289,E2 -16802.289} C_VEL
LIN {X 0,Y 306.643,Z 437.129,A -85,B 0,C 180,E1 -16802.764,E2 -16802.764} C_VEL
LIN {X 0,Y 305.527,Z 449.436,A -85,B 0,C 180,E1 -16803.442,E2 -16803.442} C_VEL
LIN {X 0,Y 304.107,Z 461.867,A -85,B 0,C 180,E1 -16804.407,E2 -16804.407} C_VEL
LIN {X 0,Y 302.313,Z 473.877,A -85,B 0,C 180,E1 -16805.629,E2 -16805.629} C_VEL
LIN {X 0,Y 300.219,Z 485.221,A -85,B 0,C 180,E1 -16807.097,E2 -16807.097} C_VEL
LIN {X 0,Y 298.311,Z 494.417,A -85,B 0,C 180,E1 -16808.582,E2 -16808.582} C_VEL
LIN {X 0,Y 296.5,Z 502.872,A -85,B 0,C 180,E1 -16810.259,E2 -16810.259} C_VEL
LIN {X 0,Y 294.578,Z 511.238,A -85,B 0,C 180,E1 -16812.315,E2 -16812.315} C_VEL
LIN {X 0,Y 292.953,Z 518.859,A -85,B 0,C 180,E1 -16814.699,E2 -16814.699} C_VEL
LIN {X 0,Y 291.65,Z 524.081,A -85,B 0,C 180,E1 -16816.766,E2 -16816.766} C_VEL
LIN {X 0,Y 290.768,Z 528.198,A -85,B 0,C 180,E1 -16818.851,E2 -16818.851} C_VEL
LIN {X 0,Y 290.37,Z 530.397,A -85,B 0,C 180,E1 -16820.246,E2 -16820.246} C_VEL
LIN {X 0,Y 290.041,Z 532.189,A -85,B 0,C 180,E1 -16821.64,E2 -16821.64} C_VEL
LIN {X 0,Y 289.608,Z 534.541,A -85,B 0,C 180,E1 -16824.43,E2 -16824.43} C_VEL
LIN {X 0,Y 289.503,Z 535.435,A -85,B 0,C 180,E1 -16827.217,E2 -16827.217} C_VEL
LIN {X 0,Y 289.445,Z 534.902,A -85,B 0,C 180,E1 -16830,E2 -16830} C_VEL
LIN {X 0,Y 289.691,Z 532.858,A -85,B 0,C 180,E1 -16832.781,E2 -16832.781} C_VEL
LIN {X 0,Y 290.294,Z 529.313,A -85,B 0,C 180,E1 -16835.557,E2 -16835.557} C_VEL
LIN {X 0,Y 291.057,Z 524.555,A -85,B 0,C 180,E1 -16838.102,E2 -16838.102} C_VEL
LIN {X 0,Y 292.058,Z 518.84,A -85,B 0,C 180,E1 -16840.397,E2 -16840.397} C_VEL
LIN {X 0,Y 293.592,Z 511.17,A -85,B 0,C 180,E1 -16842.793,E2 -16842.793} C_VEL
LIN {X 0,Y 295.219,Z 502.937,A -85,B 0,C 180,E1 -16844.827,E2 -16844.827} C_VEL
LIN {X 0,Y 296.818,Z 494.548,A -85,B 0,C 180,E1 -16846.507,E2 -16846.507} C_VEL
LIN {X 0,Y 298.402,Z 485.443,A -85,B 0,C 180,E1 -16848.006,E2 -16848.006} C_VEL
LIN {X 0,Y 299.978,Z 475.629,A -85,B 0,C 180,E1 -16849.325,E2 -16849.325} C_VEL
LIN {X 0,Y 301.767,Z 463.3,A -85,B 0,C 180,E1 -16850.625,E2 -16850.625} C_VEL
LIN {X 0,Y 303.173,Z 451.302,A -85,B 0,C 180,E1 -16851.592,E2 -16851.592} C_VEL
LIN {X 0,Y 304.262,Z 438.153,A -85,B 0,C 180,E1 -16852.369,E2 -16852.369} C_VEL
LIN {X 0,Y 305.032,Z 424.783,A -85,B 0,C 180,E1 -16852.863,E2 -16852.863} C_VEL
LIN {X 0,Y 306.803,Z 352.896,A -85,B 0,C 180,E1 -16854.464,E2 -16854.464} C_VEL
LIN {X 0,Y 301.94,Z 323.25,A -85,B 0,C 180,E1 -16855.675,E2 -16855.675} C_VEL
LIN {X 0,Y 299.57,Z 310.664,A -85,B 0,C 180,E1 -16856.266,E2 -16856.266} C_VEL
LIN {X 0,Y 299.884,Z 307.285,A -85,B 0,C 180,E1 -16857.055,E2 -16857.055} C_VEL
LIN {X 0,Y 297.882,Z 296.979,A -85,B 0,C 180,E1 -16860.089,E2 -16860.089} C_VEL
LIN {X 0,Y 295.241,Z 285.885,A -85,B 0,C 180,E1 -16863.575,E2 -16863.575} C_VEL
LIN {X 0,Y 292.147,Z 274.453,A -85,B 0,C 180,E1 -16867.451,E2 -16867.451} C_VEL
LIN {X 0,Y 291.368,Z 271.9,A -85,B 0,C 180,E1 -16868.429,E2 -16868.429} C_VEL
LIN {X 0,Y 291.32,Z 271.819,A -85,B 0,C 180,E1 -16872.491,E2 -16872.491} C_VEL
LIN {X 0,Y 291.308,Z 271.813,A -85,B 0,C 180,E1 -16876.365,E2 -16876.365} C_VEL
LIN {X 0,Y 291.322,Z 271.811,A -85,B 0,C 180,E1 -16878.498,E2 -16878.498} C_VEL
LIN {X 0,Y 290.639,Z 271.885,A -85,B 0,C 180,E1 -16879.652,E2 -16879.652} C_VEL
LIN {X 0,Y 287.787,Z 272.246,A -85,B 0,C 180,E1 -16881.533,E2 -16881.533} C_VEL
LIN {X 0,Y 285.404,Z 272.561,A -85,B 0,C 180,E1 -16883.06,E2 -16883.06} C_VEL
LIN {X 0,Y 284.42,Z 272.67,A -85,B 0,C 180,E1 -16884.243,E2 -16884.243} C_VEL
LIN {X 0,Y 284.36,Z 272.67,A -85,B 0,C 180,E1 -16884.643,E2 -16884.643} C_VEL
LIN {X 0,Y 284.294,Z 272.69,A -85,B 0,C 180,E1 -16888.725,E2 -16888.725} C_VEL
LIN {X 0,Y 284.397,Z 272.68,A -85,B 0,C 180,E1 -16892.825,E2 -16892.825} C_VEL
LIN {X 0,Y 284.363,Z 272.68,A -85,B 0,C 180,E1 -16896.706,E2 -16896.706} C_VEL
LIN {X 0,Y 284.4,Z 272.677,A -85,B 0,C 180,E1 -16901.261,E2 -16901.261} C_VEL
LIN {X 0,Y 284.474,Z 272.664,A -85,B 0,C 180,E1 -16904.469,E2 -16904.469} C_VEL
LIN {X 0,Y 284.483,Z 272.669,A -85,B 0,C 180,E1 -16908.601,E2 -16908.601} C_VEL
LIN {X 0,Y 284.635,Z 272.65,A -85,B 0,C 180,E1 -16911.48,E2 -16911.48} C_VEL
LIN {X 0,Y 284.593,Z 272.65,A -85,B 0,C 180,E1 -16914.331,E2 -16914.331} C_VEL
LIN {X 0,Y 284.85,Z 272.627,A -85,B 0,C 180,E1 -16918.586,E2 -16918.586} C_VEL
LIN {X 0,Y 284.851,Z 272.616,A -85,B 0,C 180,E1 -16921.413,E2 -16921.413} C_VEL
LIN {X 0,Y 284.693,Z 272.64,A -85,B 0,C 180,E1 -16927.09,E2 -16927.09} C_VEL
LIN {X 0,Y 284.561,Z 272.656,A -85,B 0,C 180,E1 -16929.955,E2 -16929.955} C_VEL
LIN {X 0,Y 284.473,Z 272.672,A -85,B 0,C 180,E1 -16934.303,E2 -16934.303} C_VEL
LIN {X 0,Y 284.42,Z 272.678,A -85,B 0,C 180,E1 -16937.248,E2 -16937.248} C_VEL
LIN {X 0,Y 284.374,Z 272.677,A -85,B 0,C 180,E1 -16940.242,E2 -16940.242} C_VEL
LIN {X 0,Y 284.364,Z 272.683,A -85,B 0,C 180,E1 -16943.875,E2 -16943.875} C_VEL
LIN {X 0,Y 284.393,Z 272.685,A -85,B 0,C 180,E1 -16947.174,E2 -16947.174} C_VEL
LIN {X 0,Y 284.291,Z 272.667,A -85,B 0,C 180,E1 -16951.274,E2 -16951.274} C_VEL
LIN {X 0,Y 284.337,Z 272.677,A -85,B 0,C 180,E1 -16955.348,E2 -16955.348} C_VEL
LIN {X 0,Y 284.308,Z 272.679,A -85,B 0,C 180,E1 -16958.169,E2 -16958.169} C_VEL
LIN {X 0,Y 284.265,Z 272.682,A -85,B 0,C 180,E1 -16962.125,E2 -16962.125} C_VEL
LIN {X 0,Y 284.264,Z 272.66,A -85,B 0,C 180,E1 -16966.192,E2 -16966.192} C_VEL
LIN {X 0,Y 284.315,Z 272.839,A -85,B 0,C 180,E1 -16969,E2 -16969} C_VEL
LIN {X 0,Y 287.509,Z 283.525,A -85,B 0,C 180,E1 -16972.692,E2 -16972.692} C_VEL
LIN {X 0,Y 290.377,Z 294.57,A -85,B 0,C 180,E1 -16976.175,E2 -16976.175} C_VEL
LIN {X 0,Y 291.857,Z 300.724,A -85,B 0,C 180,E1 -16977.927,E2 -16977.927} C_VEL
LIN {X 0,Y 299.171,Z 317.517,A -85,B 0,C 180,E1 -16979.224,E2 -16979.224} C_VEL
LIN {X 0,Y 301.55,Z 334.859,A -85,B 0,C 180,E1 -16979.946,E2 -16979.946} C_VEL
LIN {X 0,Y 298.408,Z 431.194,A -85,B 0,C 180,E1 -16982.329,E2 -16982.329} C_VEL
LIN {X 0,Y 297.358,Z 445.424,A -85,B 0,C 180,E1 -16982.938,E2 -16982.938} C_VEL
LIN {X 0,Y 296.08,Z 458.56,A -85,B 0,C 180,E1 -16983.763,E2 -16983.763} C_VEL
LIN {X 0,Y 294.585,Z 470.419,A -85,B 0,C 180,E1 -16984.744,E2 -16984.744} C_VEL
LIN {X 0,Y 292.843,Z 483.201,A -85,B 0,C 180,E1 -16986.11,E2 -16986.11} C_VEL
LIN {X 0,Y 290.858,Z 494.67,A -85,B 0,C 180,E1 -16987.632,E2 -16987.632} C_VEL
LIN {X 0,Y 288.94,Z 505.153,A -85,B 0,C 180,E1 -16989.349,E2 -16989.349} C_VEL
LIN {X 0,Y 287.097,Z 515.474,A -85,B 0,C 180,E1 -16991.444,E2 -16991.444} C_VEL
LIN {X 0,Y 285.486,Z 524.661,A -85,B 0,C 180,E1 -16993.758,E2 -16993.758} C_VEL
LIN {X 0,Y 284.468,Z 531.001,A -85,B 0,C 180,E1 -16995.697,E2 -16995.697} C_VEL
LIN {X 0,Y 283.526,Z 536.806,A -85,B 0,C 180,E1 -16997.837,E2 -16997.837} C_VEL
LIN {X 0,Y 282.91,Z 541.501,A -85,B 0,C 180,E1 -16999.986,E2 -16999.986} C_VEL
LIN {X 0,Y 282.556,Z 545.208,A -85,B 0,C 180,E1 -17002.137,E2 -17002.137} C_VEL
LIN {X 0,Y 282.329,Z 548.461,A -85,B 0,C 180,E1 -17004.693,E2 -17004.693} C_VEL
LIN {X 0,Y 282.33,Z 550.46,A -85,B 0,C 180,E1 -17007.146,E2 -17007.146} C_VEL
LIN {X 0,Y 282.355,Z 551.437,A -85,B 0,C 180,E1 -17010,E2 -17010} C_VEL
LIN {X 0,Y 282.331,Z 550.979,A -85,B 0,C 180,E1 -17012.854,E2 -17012.854} C_VEL
LIN {X 0,Y 282.382,Z 549.089,A -85,B 0,C 180,E1 -17015.713,E2 -17015.713} C_VEL
LIN {X 0,Y 282.682,Z 545.685,A -85,B 0,C 180,E1 -17018.579,E2 -17018.579} C_VEL
LIN {X 0,Y 283.143,Z 542.116,A -85,B 0,C 180,E1 -17020.729,E2 -17020.729} C_VEL
LIN {X 0,Y 283.956,Z 537.566,A -85,B 0,C 180,E1 -17022.871,E2 -17022.871} C_VEL
LIN {X 0,Y 285.245,Z 530.953,A -85,B 0,C 180,E1 -17025.359,E2 -17025.359} C_VEL
LIN {X 0,Y 286.866,Z 522.677,A -85,B 0,C 180,E1 -17027.833,E2 -17027.833} C_VEL
LIN {X 0,Y 288.697,Z 513.942,A -85,B 0,C 180,E1 -17029.926,E2 -17029.926} C_VEL
LIN {X 0,Y 290.902,Z 503.297,A -85,B 0,C 180,E1 -17031.991,E2 -17031.991} C_VEL
LIN {X 0,Y 293.064,Z 492.505,A -85,B 0,C 180,E1 -17033.683,E2 -17033.683} C_VEL
LIN {X 0,Y 295.007,Z 481.132,A -85,B 0,C 180,E1 -17035.139,E2 -17035.139} C_VEL
LIN {X 0,Y 296.852,Z 469.246,A -85,B 0,C 180,E1 -17036.353,E2 -17036.353} C_VEL
LIN {X 0,Y 298.62,Z 455.832,A -85,B 0,C 180,E1 -17037.413,E2 -17037.413} C_VEL
LIN {X 0,Y 300.102,Z 441.618,A -85,B 0,C 180,E1 -17038.213,E2 -17038.213} C_VEL
LIN {X 0,Y 301.072,Z 427.614,A -85,B 0,C 180,E1 -17038.732,E2 -17038.732} C_VEL
LIN {X 0,Y 304.201,Z 336.146,A -85,B 0,C 180,E1 -17040.967,E2 -17040.967} C_VEL
LIN {X 0,Y 301.995,Z 321.643,A -85,B 0,C 180,E1 -17041.624,E2 -17041.624} C_VEL
LIN {X 0,Y 293.638,Z 303.668,A -85,B 0,C 180,E1 -17043.147,E2 -17043.147} C_VEL
LIN {X 0,Y 292.217,Z 300.515,A -85,B 0,C 180,E1 -17043.485,E2 -17043.485} C_VEL
LIN {X 0,Y 289.902,Z 291.42,A -85,B 0,C 180,E1 -17046.334,E2 -17046.334} C_VEL
LIN {X 0,Y 286.873,Z 280.801,A -85,B 0,C 180,E1 -17049.975,E2 -17049.975} C_VEL
LIN {X 0,Y 284.35,Z 272.76,A -85,B 0,C 180,E1 -17053.04,E2 -17053.04} C_VEL
LIN {X 0,Y 284.295,Z 272.696,A -85,B 0,C 180,E1 -17056.197,E2 -17056.197} C_VEL
LIN {X 0,Y 284.304,Z 272.682,A -85,B 0,C 180,E1 -17060.024,E2 -17060.024} C_VEL
LIN {X 0,Y 284.333,Z 272.665,A -85,B 0,C 180,E1 -17063.614,E2 -17063.614} C_VEL
LIN {X 0,Y 284.304,Z 272.697,A -85,B 0,C 180,E1 -17067.189,E2 -17067.189} C_VEL
LIN {X 0,Y 284.354,Z 272.654,A -85,B 0,C 180,E1 -17070.376,E2 -17070.376} C_VEL
LIN {X 0,Y 284.374,Z 272.688,A -85,B 0,C 180,E1 -17073.587,E2 -17073.587} C_VEL
LIN {X 0,Y 284.362,Z 272.687,A -85,B 0,C 180,E1 -17076.707,E2 -17076.707} C_VEL
LIN {X 0,Y 284.399,Z 272.683,A -85,B 0,C 180,E1 -17081.262,E2 -17081.262} C_VEL
LIN {X 0,Y 284.488,Z 272.664,A -85,B 0,C 180,E1 -17084.46,E2 -17084.46} C_VEL
LIN {X 0,Y 284.483,Z 272.662,A -85,B 0,C 180,E1 -17088.602,E2 -17088.602} C_VEL
LIN {X 0,Y 284.652,Z 272.646,A -85,B 0,C 180,E1 -17091.481,E2 -17091.481} C_VEL
LIN {X 0,Y 284.595,Z 272.658,A -85,B 0,C 180,E1 -17094.332,E2 -17094.332} C_VEL
LIN {X 0,Y 284.851,Z 272.621,A -85,B 0,C 180,E1 -17098.587,E2 -17098.587} C_VEL
LIN {X 0,Y 284.851,Z 272.618,A -85,B 0,C 180,E1 -17101.414,E2 -17101.414} C_VEL
LIN {X 0,Y 284.694,Z 272.635,A -85,B 0,C 180,E1 -17107.091,E2 -17107.091} C_VEL
LIN {X 0,Y 284.563,Z 272.661,A -85,B 0,C 180,E1 -17109.956,E2 -17109.956} C_VEL
LIN {X 0,Y 284.475,Z 272.673,A -85,B 0,C 180,E1 -17114.304,E2 -17114.304} C_VEL
LIN {X 0,Y 284.422,Z 272.678,A -85,B 0,C 180,E1 -17117.249,E2 -17117.249} C_VEL
LIN {X 0,Y 284.378,Z 272.676,A -85,B 0,C 180,E1 -17120.243,E2 -17120.243} C_VEL
LIN {X 0,Y 284.366,Z 272.68,A -85,B 0,C 180,E1 -17123.876,E2 -17123.876} C_VEL
LIN {X 0,Y 284.394,Z 272.671,A -85,B 0,C 180,E1 -17127.174,E2 -17127.174} C_VEL
LIN {X 0,Y 284.292,Z 272.691,A -85,B 0,C 180,E1 -17131.275,E2 -17131.275} C_VEL
LIN {X 0,Y 284.36,Z 272.664,A -85,B 0,C 180,E1 -17135.355,E2 -17135.355} C_VEL
LIN {X 0,Y 284.322,Z 272.69,A -85,B 0,C 180,E1 -17138.168,E2 -17138.168} C_VEL
LIN {X 0,Y 284.27,Z 272.702,A -85,B 0,C 180,E1 -17142.126,E2 -17142.126} C_VEL
LIN {X 0,Y 284.287,Z 272.849,A -85,B 0,C 180,E1 -17144.821,E2 -17144.821} C_VEL
LIN {X 0,Y 286.92,Z 281.443,A -85,B 0,C 180,E1 -17148.208,E2 -17148.208} C_VEL
LIN {X 0,Y 289.431,Z 290.544,A -85,B 0,C 180,E1 -17151.49,E2 -17151.49} C_VEL
LIN {X 0,Y 291.429,Z 298.622,A -85,B 0,C 180,E1 -17154.212,E2 -17154.212} C_VEL
LIN {X 0,Y 293.892,Z 310.241,A -85,B 0,C 180,E1 -17157.813,E2 -17157.813} C_VEL
LIN {X 0,Y 295.803,Z 315.113,A -85,B 0,C 180,E1 -17158.222,E2 -17158.222} C_VEL
LIN {X 0,Y 300.693,Z 340.55,A -85,B 0,C 180,E1 -17159.469,E2 -17159.469} C_VEL
LIN {X 0,Y 303.25,Z 355.855,A -85,B 0,C 180,E1 -17160.15,E2 -17160.15} C_VEL
LIN {X 0,Y 301.152,Z 425.361,A -85,B 0,C 180,E1 -17161.707,E2 -17161.707} C_VEL
LIN {X 0,Y 300.204,Z 438.959,A -85,B 0,C 180,E1 -17162.224,E2 -17162.224} C_VEL
LIN {X 0,Y 299.068,Z 450.693,A -85,B 0,C 180,E1 -17162.916,E2 -17162.916} C_VEL
LIN {X 0,Y 297.619,Z 462.713,A -85,B 0,C 180,E1 -17163.888,E2 -17163.888} C_VEL
LIN {X 0,Y 295.862,Z 473.974,A -85,B 0,C 180,E1 -17165.062,E2 -17165.062} C_VEL
LIN {X 0,Y 293.692,Z 485.323,A -85,B 0,C 180,E1 -17166.558,E2 -17166.558} C_VEL
LIN {X 0,Y 291.698,Z 494.526,A -85,B 0,C 180,E1 -17168.072,E2 -17168.072} C_VEL
LIN {X 0,Y 289.802,Z 502.99,A -85,B 0,C 180,E1 -17169.783,E2 -17169.783} C_VEL
LIN {X 0,Y 287.803,Z 511.288,A -85,B 0,C 180,E1 -17171.86,E2 -17171.86} C_VEL
LIN {X 0,Y 286.467,Z 517.013,A -85,B 0,C 180,E1 -17173.613,E2 -17173.613} C_VEL
LIN {X 0,Y 285.173,Z 522.641,A -85,B 0,C 180,E1 -17175.733,E2 -17175.733} C_VEL
LIN {X 0,Y 284.042,Z 527.117,A -85,B 0,C 180,E1 -17177.859,E2 -17177.859} C_VEL
LIN {X 0,Y 283.346,Z 530.561,A -85,B 0,C 180,E1 -17180.001,E2 -17180.001} C_VEL
LIN {X 0,Y 283.002,Z 532.359,A -85,B 0,C 180,E1 -17181.431,E2 -17181.431} C_VEL
LIN {X 0,Y 282.526,Z 534.725,A -85,B 0,C 180,E1 -17184.29,E2 -17184.29} C_VEL
LIN {X 0,Y 282.433,Z 535.631,A -85,B 0,C 180,E1 -17187.147,E2 -17187.147} C_VEL
LIN {X 0,Y 282.365,Z 535.114,A -85,B 0,C 180,E1 -17190,E2 -17190} C_VEL
LIN {X 0,Y 282.622,Z 533.085,A -85,B 0,C 180,E1 -17192.851,E2 -17192.851} C_VEL
LIN {X 0,Y 283.237,Z 529.555,A -85,B 0,C 180,E1 -17195.696,E2 -17195.696} C_VEL
LIN {X 0,Y 283.966,Z 525.227,A -85,B 0,C 180,E1 -17198.114,E2 -17198.114} C_VEL
LIN {X 0,Y 285.089,Z 519.129,A -85,B 0,C 180,E1 -17200.654,E2 -17200.654} C_VEL
LIN {X 0,Y 286.702,Z 511.482,A -85,B 0,C 180,E1 -17203.105,E2 -17203.105} C_VEL
LIN {X 0,Y 288.384,Z 503.286,A -85,B 0,C 180,E1 -17205.187,E2 -17205.187} C_VEL
LIN {X 0,Y 290.025,Z 494.94,A -85,B 0,C 180,E1 -17206.905,E2 -17206.905} C_VEL
LIN {X 0,Y 291.917,Z 484.738,A -85,B 0,C 180,E1 -17208.602,E2 -17208.602} C_VEL
LIN {X 0,Y 293.717,Z 473.332,A -85,B 0,C 180,E1 -17210.118,E2 -17210.118} C_VEL
LIN {X 0,Y 295.389,Z 462.173,A -85,B 0,C 180,E1 -17211.274,E2 -17211.274} C_VEL
LIN {X 0,Y 296.871,Z 449.818,A -85,B 0,C 180,E1 -17212.257,E2 -17212.257} C_VEL
LIN {X 0,Y 297.9,Z 436.727,A -85,B 0,C 180,E1 -17213.007,E2 -17213.007} C_VEL
LIN {X 0,Y 298.715,Z 422.885,A -85,B 0,C 180,E1 -17213.491,E2 -17213.491} C_VEL
LIN {X 0,Y 300.448,Z 353.747,A -85,B 0,C 180,E1 -17215.058,E2 -17215.058} C_VEL
LIN {X 0,Y 295.937,Z 325.751,A -85,B 0,C 180,E1 -17216.235,E2 -17216.235} C_VEL
LIN {X 0,Y 293.057,Z 310.596,A -85,B 0,C 180,E1 -17216.965,E2 -17216.965} C_VEL
LIN {X 0,Y 292.996,Z 308.531,A -85,B 0,C 180,E1 -17217.437,E2 -17217.437} C_VEL
LIN {X 0,Y 291.02,Z 298.505,A -85,B 0,C 180,E1 -17220.473,E2 -17220.473} C_VEL
LIN {X 0,Y 288.329,Z 287.302,A -85,B 0,C 180,E1 -17224.098,E2 -17224.098} C_VEL
LIN {X 0,Y 285.746,Z 277.465,A -85,B 0,C 180,E1 -17227.514,E2 -17227.514} C_VEL
LIN {X 0,Y 284.334,Z 272.738,A -85,B 0,C 180,E1 -17229.356,E2 -17229.356} C_VEL
LIN {X 0,Y 284.255,Z 272.693,A -85,B 0,C 180,E1 -17233.81,E2 -17233.81} C_VEL
LIN {X 0,Y 284.271,Z 272.696,A -85,B 0,C 180,E1 -17238.123,E2 -17238.123} C_VEL
LIN {X 0,Y 284.333,Z 272.69,A -85,B 0,C 180,E1 -17242.274,E2 -17242.274} C_VEL
LIN {X 0,Y 284.36,Z 272.67,A -85,B 0,C 180,E1 -17244.643,E2 -17244.643} C_VEL
LIN {X 0,Y 283.725,Z 272.742,A -85,B 0,C 180,E1 -17245.824,E2 -17245.824} C_VEL
LIN {X 0,Y 280.818,Z 273.109,A -85,B 0,C 180,E1 -17247.745,E2 -17247.745} C_VEL
LIN {X 0,Y 278.345,Z 273.438,A -85,B 0,C 180,E1 -17249.306,E2 -17249.306} C_VEL
LIN {X 0,Y 277.316,Z 273.565,A -85,B 0,C 180,E1 -17250.518,E2 -17250.518} C_VEL
LIN {X 0,Y 277.252,Z 273.565,A -85,B 0,C 180,E1 -17250.928,E2 -17250.928} C_VEL
LIN {X 0,Y 277.359,Z 273.556,A -85,B 0,C 180,E1 -17252.863,E2 -17252.863} C_VEL
LIN {X 0,Y 277.325,Z 273.553,A -85,B 0,C 180,E1 -17256.079,E2 -17256.079} C_VEL
LIN {X 0,Y 277.341,Z 273.552,A -85,B 0,C 180,E1 -17260.765,E2 -17260.765} C_VEL
LIN {X 0,Y 277.424,Z 273.54,A -85,B 0,C 180,E1 -17265.325,E2 -17265.325} C_VEL
LIN {X 0,Y 277.457,Z 273.535,A -85,B 0,C 180,E1 -17269.786,E2 -17269.786} C_VEL
LIN {X 0,Y 277.636,Z 273.528,A -85,B 0,C 180,E1 -17272.728,E2 -17272.728} C_VEL
LIN {X 0,Y 277.816,Z 273.503,A -85,B 0,C 180,E1 -17278.55,E2 -17278.55} C_VEL
LIN {X 0,Y 277.816,Z 273.492,A -85,B 0,C 180,E1 -17281.449,E2 -17281.449} C_VEL
LIN {X 0,Y 277.648,Z 273.519,A -85,B 0,C 180,E1 -17287.271,E2 -17287.271} C_VEL
LIN {X 0,Y 277.502,Z 273.532,A -85,B 0,C 180,E1 -17290.211,E2 -17290.211} C_VEL
LIN {X 0,Y 277.423,Z 273.547,A -85,B 0,C 180,E1 -17294.674,E2 -17294.674} C_VEL
LIN {X 0,Y 277.34,Z 273.561,A -85,B 0,C 180,E1 -17299.234,E2 -17299.234} C_VEL
LIN {X 0,Y 277.314,Z 273.558,A -85,B 0,C 180,E1 -17304.17,E2 -17304.17} C_VEL
LIN {X 0,Y 277.321,Z 273.563,A -85,B 0,C 180,E1 -17307.505,E2 -17307.505} C_VEL
LIN {X 0,Y 277.268,Z 273.537,A -85,B 0,C 180,E1 -17310.482,E2 -17310.482} C_VEL
LIN {X 0,Y 277.243,Z 273.579,A -85,B 0,C 180,E1 -17313.896,E2 -17313.896} C_VEL
LIN {X 0,Y 277.263,Z 273.548,A -85,B 0,C 180,E1 -17317.47,E2 -17317.47} C_VEL
LIN {X 0,Y 277.205,Z 273.565,A -85,B 0,C 180,E1 -17321.237,E2 -17321.237} C_VEL
LIN {X 0,Y 277.213,Z 273.562,A -85,B 0,C 180,E1 -17325.224,E2 -17325.224} C_VEL
LIN {X 0,Y 277.27,Z 273.722,A -85,B 0,C 180,E1 -17328.037,E2 -17328.037} C_VEL
LIN {X 0,Y 280.217,Z 283.591,A -85,B 0,C 180,E1 -17331.606,E2 -17331.606} C_VEL
LIN {X 0,Y 282.767,Z 292.911,A -85,B 0,C 180,E1 -17334.701,E2 -17334.701} C_VEL
LIN {X 0,Y 284.663,Z 300.687,A -85,B 0,C 180,E1 -17337.079,E2 -17337.079} C_VEL
LIN {X 0,Y 292.455,Z 318.355,A -85,B 0,C 180,E1 -17338.529,E2 -17338.529} C_VEL
LIN {X 0,Y 293.247,Z 320.771,A -85,B 0,C 180,E1 -17338.685,E2 -17338.685} C_VEL
LIN {X 0,Y 295.293,Z 336.741,A -85,B 0,C 180,E1 -17339.356,E2 -17339.356} C_VEL
LIN {X 0,Y 292.039,Z 430.949,A -85,B 0,C 180,E1 -17341.72,E2 -17341.72} C_VEL
LIN {X 0,Y 290.944,Z 445.241,A -85,B 0,C 180,E1 -17342.339,E2 -17342.339} C_VEL
LIN {X 0,Y 289.667,Z 457.837,A -85,B 0,C 180,E1 -17343.136,E2 -17343.136} C_VEL
LIN {X 0,Y 288.11,Z 470.021,A -85,B 0,C 180,E1 -17344.156,E2 -17344.156} C_VEL
LIN {X 0,Y 286.29,Z 482.704,A -85,B 0,C 180,E1 -17345.528,E2 -17345.528} C_VEL
LIN {X 0,Y 284.279,Z 494.24,A -85,B 0,C 180,E1 -17347.085,E2 -17347.085} C_VEL
LIN {X 0,Y 282.237,Z 504.77,A -85,B 0,C 180,E1 -17348.835,E2 -17348.835} C_VEL
LIN {X 0,Y 280.299,Z 515.145,A -85,B 0,C 180,E1 -17350.977,E2 -17350.977} C_VEL
LIN {X 0,Y 278.818,Z 523.54,A -85,B 0,C 180,E1 -17353.112,E2 -17353.112} C_VEL
LIN {X 0,Y 277.533,Z 530.721,A -85,B 0,C 180,E1 -17355.332,E2 -17355.332} C_VEL
LIN {X 0,Y 276.537,Z 536.543,A -85,B 0,C 180,E1 -17357.525,E2 -17357.525} C_VEL
LIN {X 0,Y 275.864,Z 541.247,A -85,B 0,C 180,E1 -17359.728,E2 -17359.728} C_VEL
LIN {X 0,Y 275.49,Z 544.97,A -85,B 0,C 180,E1 -17361.934,E2 -17361.934} C_VEL
LIN {X 0,Y 275.231,Z 548.469,A -85,B 0,C 180,E1 -17364.784,E2 -17364.784} C_VEL
LIN {X 0,Y 275.238,Z 550.248,A -85,B 0,C 180,E1 -17367.073,E2 -17367.073} C_VEL
LIN {X 0,Y 275.259,Z 550.921,A -85,B 0,C 180,E1 -17368.537,E2 -17368.537} C_VEL
LIN {X 0,Y 275.276,Z 551.236,A -85,B 0,C 180,E1 -17370,E2 -17370} C_VEL
LIN {X 0,Y 275.259,Z 551.19,A -85,B 0,C 180,E1 -17371.463,E2 -17371.463} C_VEL
LIN {X 0,Y 275.24,Z 550.788,A -85,B 0,C 180,E1 -17372.927,E2 -17372.927} C_VEL
LIN {X 0,Y 275.294,Z 548.907,A -85,B 0,C 180,E1 -17375.861,E2 -17375.861} C_VEL
LIN {X 0,Y 275.634,Z 545.514,A -85,B 0,C 180,E1 -17378.8,E2 -17378.8} C_VEL
LIN {X 0,Y 276.335,Z 540.529,A -85,B 0,C 180,E1 -17381.739,E2 -17381.739} C_VEL
LIN {X 0,Y 277.351,Z 535.68,A -85,B 0,C 180,E1 -17383.929,E2 -17383.929} C_VEL
LIN {X 0,Y 278.821,Z 528.542,A -85,B 0,C 180,E1 -17386.494,E2 -17386.494} C_VEL
LIN {X 0,Y 280.635,Z 519.783,A -85,B 0,C 180,E1 -17388.999,E2 -17388.999} C_VEL
LIN {X 0,Y 282.702,Z 510.507,A -85,B 0,C 180,E1 -17391.129,E2 -17391.129} C_VEL
LIN {X 0,Y 284.947,Z 500.181,A -85,B 0,C 180,E1 -17393.05,E2 -17393.05} C_VEL
LIN {X 0,Y 287.325,Z 488.52,A -85,B 0,C 180,E1 -17394.789,E2 -17394.789} C_VEL
LIN {X 0,Y 289.192,Z 477.482,A -85,B 0,C 180,E1 -17396.134,E2 -17396.134} C_VEL
LIN {X 0,Y 291.041,Z 465.318,A -85,B 0,C 180,E1 -17397.31,E2 -17397.31} C_VEL
LIN {X 0,Y 292.81,Z 451.828,A -85,B 0,C 180,E1 -17398.296,E2 -17398.296} C_VEL
LIN {X 0,Y 294.225,Z 437.808,A -85,B 0,C 180,E1 -17399.025,E2 -17399.025} C_VEL
LIN {X 0,Y 295.008,Z 424.391,A -85,B 0,C 180,E1 -17399.478,E2 -17399.478} C_VEL
LIN {X 0,Y 298.07,Z 337.093,A -85,B 0,C 180,E1 -17401.637,E2 -17401.637} C_VEL
LIN {X 0,Y 296.08,Z 324.136,A -85,B 0,C 180,E1 -17402.247,E2 -17402.247} C_VEL
LIN {X 0,Y 287.945,Z 306.706,A -85,B 0,C 180,E1 -17403.785,E2 -17403.785} C_VEL
LIN {X 0,Y 285.119,Z 300.708,A -85,B 0,C 180,E1 -17404.406,E2 -17404.406} C_VEL
LIN {X 0,Y 282.415,Z 290.58,A -85,B 0,C 180,E1 -17407.749,E2 -17407.749} C_VEL
LIN {X 0,Y 279.718,Z 281.338,A -85,B 0,C 180,E1 -17411.083,E2 -17411.083} C_VEL
LIN {X 0,Y 277.277,Z 273.641,A -85,B 0,C 180,E1 -17414.183,E2 -17414.183} C_VEL
LIN {X 0,Y 277.229,Z 273.566,A -85,B 0,C 180,E1 -17417.321,E2 -17417.321} C_VEL
LIN {X 0,Y 277.268,Z 273.569,A -85,B 0,C 180,E1 -17421.79,E2 -17421.79} C_VEL
LIN {X 0,Y 277.282,Z 273.543,A -85,B 0,C 180,E1 -17424.342,E2 -17424.342} C_VEL
LIN {X 0,Y 277.241,Z 273.568,A -85,B 0,C 180,E1 -17427.836,E2 -17427.836} C_VEL
LIN {X 0,Y 277.267,Z 273.542,A -85,B 0,C 180,E1 -17431.21,E2 -17431.21} C_VEL
LIN {X 0,Y 277.31,Z 273.564,A -85,B 0,C 180,E1 -17434.48,E2 -17434.48} C_VEL
LIN {X 0,Y 277.281,Z 273.573,A -85,B 0,C 180,E1 -17437.655,E2 -17437.655} C_VEL
LIN {X 0,Y 277.341,Z 273.561,A -85,B 0,C 180,E1 -17440.766,E2 -17440.766} C_VEL
LIN {X 0,Y 277.43,Z 273.549,A -85,B 0,C 180,E1 -17445.326,E2 -17445.326} C_VEL
LIN {X 0,Y 277.502,Z 273.54,A -85,B 0,C 180,E1 -17449.789,E2 -17449.789} C_VEL
LIN {X 0,Y 277.645,Z 273.511,A -85,B 0,C 180,E1 -17452.729,E2 -17452.729} C_VEL
LIN {X 0,Y 277.817,Z 273.497,A -85,B 0,C 180,E1 -17458.551,E2 -17458.551} C_VEL
LIN {X 0,Y 277.817,Z 273.493,A -85,B 0,C 180,E1 -17461.45,E2 -17461.45} C_VEL
LIN {X 0,Y 277.649,Z 273.512,A -85,B 0,C 180,E1 -17467.272,E2 -17467.272} C_VEL
LIN {X 0,Y 277.503,Z 273.539,A -85,B 0,C 180,E1 -17470.212,E2 -17470.212} C_VEL
LIN {X 0,Y 277.425,Z 273.548,A -85,B 0,C 180,E1 -17474.675,E2 -17474.675} C_VEL
LIN {X 0,Y 277.342,Z 273.555,A -85,B 0,C 180,E1 -17479.235,E2 -17479.235} C_VEL
LIN {X 0,Y 277.326,Z 273.556,A -85,B 0,C 180,E1 -17483.921,E2 -17483.921} C_VEL
LIN {X 0,Y 277.322,Z 273.544,A -85,B 0,C 180,E1 -17487.505,E2 -17487.505} C_VEL
LIN {X 0,Y 277.271,Z 273.549,A -85,B 0,C 180,E1 -17490.482,E2 -17490.482} C_VEL
LIN {X 0,Y 277.253,Z 273.555,A -85,B 0,C 180,E1 -17493.896,E2 -17493.896} C_VEL
LIN {X 0,Y 277.281,Z 273.572,A -85,B 0,C 180,E1 -17497.468,E2 -17497.468} C_VEL
LIN {X 0,Y 277.21,Z 273.566,A -85,B 0,C 180,E1 -17501.237,E2 -17501.237} C_VEL
LIN {X 0,Y 277.242,Z 273.76,A -85,B 0,C 180,E1 -17503.736,E2 -17503.736} C_VEL
LIN {X 0,Y 279.932,Z 282.501,A -85,B 0,C 180,E1 -17507.324,E2 -17507.324} C_VEL
LIN {X 0,Y 282.606,Z 291.946,A -85,B 0,C 180,E1 -17510.871,E2 -17510.871} C_VEL
LIN {X 0,Y 284.59,Z 299.932,A -85,B 0,C 180,E1 -17513.653,E2 -17513.653} C_VEL
LIN {X 0,Y 286.72,Z 310.024,A -85,B 0,C 180,E1 -17516.883,E2 -17516.883} C_VEL
LIN {X 0,Y 289.993,Z 317.363,A -85,B 0,C 180,E1 -17517.563,E2 -17517.563} C_VEL
LIN {X 0,Y 294.734,Z 342.365,A -85,B 0,C 180,E1 -17518.824,E2 -17518.824} C_VEL
LIN {X 0,Y 297.094,Z 356.504,A -85,B 0,C 180,E1 -17519.475,E2 -17519.475} C_VEL
LIN {X 0,Y 294.848,Z 427.12,A -85,B 0,C 180,E1 -17521.1,E2 -17521.1} C_VEL
LIN {X 0,Y 293.776,Z 440.607,A -85,B 0,C 180,E1 -17521.659,E2 -17521.659} C_VEL
LIN {X 0,Y 292.487,Z 453.061,A -85,B 0,C 180,E1 -17522.449,E2 -17522.449} C_VEL
LIN {X 0,Y 290.873,Z 465.498,A -85,B 0,C 180,E1 -17523.529,E2 -17523.529} C_VEL
LIN {X 0,Y 288.945,Z 476.858,A -85,B 0,C 180,E1 -17524.809,E2 -17524.809} C_VEL
LIN {X 0,Y 286.708,Z 487.602,A -85,B 0,C 180,E1 -17526.335,E2 -17526.335} C_VEL
LIN {X 0,Y 284.705,Z 496.433,A -85,B 0,C 180,E1 -17527.886,E2 -17527.886} C_VEL
LIN {X 0,Y 282.373,Z 506.056,A -85,B 0,C 180,E1 -17529.988,E2 -17529.988} C_VEL
LIN {X 0,Y 280.391,Z 513.958,A -85,B 0,C 180,E1 -17532.157,E2 -17532.157} C_VEL
LIN {X 0,Y 278.736,Z 521.017,A -85,B 0,C 180,E1 -17534.648,E2 -17534.648} C_VEL
LIN {X 0,Y 277.37,Z 525.882,A -85,B 0,C 180,E1 -17536.818,E2 -17536.818} C_VEL
LIN {X 0,Y 276.541,Z 529.69,A -85,B 0,C 180,E1 -17539.012,E2 -17539.012} C_VEL
LIN {X 0,Y 275.959,Z 532.53,A -85,B 0,C 180,E1 -17541.211,E2 -17541.211} C_VEL
LIN {X 0,Y 275.452,Z 534.91,A -85,B 0,C 180,E1 -17544.142,E2 -17544.142} C_VEL
LIN {X 0,Y 275.341,Z 535.827,A -85,B 0,C 180,E1 -17547.074,E2 -17547.074} C_VEL
LIN {X 0,Y 275.287,Z 535.325,A -85,B 0,C 180,E1 -17550,E2 -17550} C_VEL
LIN {X 0,Y 275.555,Z 533.312,A -85,B 0,C 180,E1 -17552.924,E2 -17552.924} C_VEL
LIN {X 0,Y 275.857,Z 531.746,A -85,B 0,C 180,E1 -17554.383,E2 -17554.383} C_VEL
LIN {X 0,Y 276.394,Z 528.648,A -85,B 0,C 180,E1 -17556.57,E2 -17556.57} C_VEL
LIN {X 0,Y 277.113,Z 524.577,A -85,B 0,C 180,E1 -17558.752,E2 -17558.752} C_VEL
LIN {X 0,Y 278.141,Z 519.416,A -85,B 0,C 180,E1 -17560.924,E2 -17560.924} C_VEL
LIN {X 0,Y 279.796,Z 511.794,A -85,B 0,C 180,E1 -17563.435,E2 -17563.435} C_VEL
LIN {X 0,Y 281.561,Z 503.629,A -85,B 0,C 180,E1 -17565.564,E2 -17565.564} C_VEL
LIN {X 0,Y 283.26,Z 495.324,A -85,B 0,C 180,E1 -17567.321,E2 -17567.321} C_VEL
LIN {X 0,Y 285.219,Z 485.192,A -85,B 0,C 180,E1 -17569.055,E2 -17569.055} C_VEL
LIN {X 0,Y 287.096,Z 473.857,A -85,B 0,C 180,E1 -17570.603,E2 -17570.603} C_VEL
LIN {X 0,Y 288.831,Z 462.8,A -85,B 0,C 180,E1 -17571.781,E2 -17571.781} C_VEL
LIN {X 0,Y 290.349,Z 450.606,A -85,B 0,C 180,E1 -17572.785,E2 -17572.785} C_VEL
LIN {X 0,Y 291.432,Z 437.515,A -85,B 0,C 180,E1 -17573.571,E2 -17573.571} C_VEL
LIN {X 0,Y 292.269,Z 424.575,A -85,B 0,C 180,E1 -17574.053,E2 -17574.053} C_VEL
LIN {X 0,Y 294.106,Z 354.131,A -85,B 0,C 180,E1 -17575.692,E2 -17575.692} C_VEL
LIN {X 0,Y 289.094,Z 323.391,A -85,B 0,C 180,E1 -17577.042,E2 -17577.042} C_VEL
LIN {X 0,Y 286.553,Z 311.279,A -85,B 0,C 180,E1 -17577.662,E2 -17577.662} C_VEL
LIN {X 0,Y 286.146,Z 309.824,A -85,B 0,C 180,E1 -17577.846,E2 -17577.846} C_VEL
LIN {X 0,Y 284.102,Z 299.762,A -85,B 0,C 180,E1 -17580.963,E2 -17580.963} C_VEL
LIN {X 0,Y 281.565,Z 289.015,A -85,B 0,C 180,E1 -17584.542,E2 -17584.542} C_VEL
LIN {X 0,Y 278.959,Z 279.326,A -85,B 0,C 180,E1 -17588.023,E2 -17588.023} C_VEL
LIN {X 0,Y 277.245,Z 273.635,A -85,B 0,C 180,E1 -17590.279,E2 -17590.279} C_VEL
LIN {X 0,Y 277.209,Z 273.58,A -85,B 0,C 180,E1 -17593.197,E2 -17593.197} C_VEL
LIN {X 0,Y 277.214,Z 273.58,A -85,B 0,C 180,E1 -17597.324,E2 -17597.324} C_VEL
LIN {X 0,Y 277.273,Z 273.558,A -85,B 0,C 180,E1 -17601.789,E2 -17601.789} C_VEL
LIN {X 0,Y 277.277,Z 273.552,A -85,B 0,C 180,E1 -17604.62,E2 -17604.62} C_VEL
LIN {X 0,Y 277.243,Z 273.553,A -85,B 0,C 180,E1 -17607.835,E2 -17607.835} C_VEL
LIN {X 0,Y 277.252,Z 273.565,A -85,B 0,C 180,E1 -17610.928,E2 -17610.928} C_VEL
LIN {X 0,Y 276.641,Z 273.644,A -85,B 0,C 180,E1 -17612.141,E2 -17612.141} C_VEL
LIN {X 0,Y 273.821,Z 274.002,A -85,B 0,C 180,E1 -17614.117,E2 -17614.117} C_VEL
LIN {X 0,Y 271.38,Z 274.304,A -85,B 0,C 180,E1 -17615.722,E2 -17615.722} C_VEL
LIN {X 0,Y 270.308,Z 274.433,A -85,B 0,C 180,E1 -17616.966,E2 -17616.966} C_VEL
LIN {X 0,Y 270.209,Z 274.445,A -85,B 0,C 180,E1 -17617.388,E2 -17617.388} C_VEL
LIN {X 0,Y 270.298,Z 274.428,A -85,B 0,C 180,E1 -17620.244,E2 -17620.244} C_VEL
LIN {X 0,Y 270.393,Z 274.415,A -85,B 0,C 180,E1 -17624.934,E2 -17624.934} C_VEL
LIN {X 0,Y 270.409,Z 274.414,A -85,B 0,C 180,E1 -17629.517,E2 -17629.517} C_VEL
LIN {X 0,Y 270.594,Z 274.405,A -85,B 0,C 180,E1 -17632.538,E2 -17632.538} C_VEL
LIN {X 0,Y 270.782,Z 274.38,A -85,B 0,C 180,E1 -17638.512,E2 -17638.512} C_VEL
LIN {X 0,Y 270.782,Z 274.368,A -85,B 0,C 180,E1 -17641.487,E2 -17641.487} C_VEL
LIN {X 0,Y 270.606,Z 274.398,A -85,B 0,C 180,E1 -17647.461,E2 -17647.461} C_VEL
LIN {X 0,Y 270.437,Z 274.41,A -85,B 0,C 180,E1 -17650.481,E2 -17650.481} C_VEL
LIN {X 0,Y 270.391,Z 274.421,A -85,B 0,C 180,E1 -17655.065,E2 -17655.065} C_VEL
LIN {X 0,Y 270.297,Z 274.433,A -85,B 0,C 180,E1 -17659.755,E2 -17659.755} C_VEL
LIN {X 0,Y 270.27,Z 274.434,A -85,B 0,C 180,E1 -17664.586,E2 -17664.586} C_VEL
LIN {X 0,Y 270.266,Z 274.436,A -85,B 0,C 180,E1 -17667.909,E2 -17667.909} C_VEL
LIN {X 0,Y 270.18,Z 274.424,A -85,B 0,C 180,E1 -17671.348,E2 -17671.348} C_VEL
LIN {X 0,Y 270.198,Z 274.444,A -85,B 0,C 180,E1 -17674.906,E2 -17674.906} C_VEL
LIN {X 0,Y 270.194,Z 274.445,A -85,B 0,C 180,E1 -17678.711,E2 -17678.711} C_VEL
LIN {X 0,Y 270.168,Z 274.443,A -85,B 0,C 180,E1 -17683.251,E2 -17683.251} C_VEL
LIN {X 0,Y 270.201,Z 274.647,A -85,B 0,C 180,E1 -17687.027,E2 -17687.027} C_VEL
LIN {X 0,Y 273.069,Z 283.895,A -85,B 0,C 180,E1 -17690.544,E2 -17690.544} C_VEL
LIN {X 0,Y 275.927,Z 294.317,A -85,B 0,C 180,E1 -17694.14,E2 -17694.14} C_VEL
LIN {X 0,Y 277.579,Z 300.985,A -85,B 0,C 180,E1 -17696.23,E2 -17696.23} C_VEL
LIN {X 0,Y 286.088,Z 319.953,A -85,B 0,C 180,E1 -17697.86,E2 -17697.86} C_VEL
LIN {X 0,Y 287.217,Z 322.993,A -85,B 0,C 180,E1 -17698.079,E2 -17698.079} C_VEL
LIN {X 0,Y 289.053,Z 337.383,A -85,B 0,C 180,E1 -17698.703,E2 -17698.703} C_VEL
LIN {X 0,Y 285.71,Z 430.702,A -85,B 0,C 180,E1 -17701.086,E2 -17701.086} C_VEL
LIN {X 0,Y 284.558,Z 445.055,A -85,B 0,C 180,E1 -17701.713,E2 -17701.713} C_VEL
LIN {X 0,Y 283.193,Z 458.249,A -85,B 0,C 180,E1 -17702.571,E2 -17702.571} C_VEL
LIN {X 0,Y 281.414,Z 471.511,A -85,B 0,C 180,E1 -17703.727,E2 -17703.727} C_VEL
LIN {X 0,Y 279.588,Z 483.65,A -85,B 0,C 180,E1 -17705.1,E2 -17705.1} C_VEL
LIN {X 0,Y 277.487,Z 494.996,A -85,B 0,C 180,E1 -17706.688,E2 -17706.688} C_VEL
LIN {X 0,Y 275.568,Z 504.387,A -85,B 0,C 180,E1 -17708.297,E2 -17708.297} C_VEL
LIN {X 0,Y 273.541,Z 514.816,A -85,B 0,C 180,E1 -17710.488,E2 -17710.488} C_VEL
LIN {X 0,Y 271.883,Z 523.616,A -85,B 0,C 180,E1 -17712.784,E2 -17712.784} C_VEL
LIN {X 0,Y 270.629,Z 530.442,A -85,B 0,C 180,E1 -17714.949,E2 -17714.949} C_VEL
LIN {X 0,Y 269.564,Z 536.279,A -85,B 0,C 180,E1 -17717.197,E2 -17717.197} C_VEL
LIN {X 0,Y 268.837,Z 540.994,A -85,B 0,C 180,E1 -17719.456,E2 -17719.456} C_VEL
LIN {X 0,Y 268.444,Z 544.733,A -85,B 0,C 180,E1 -17721.721,E2 -17721.721} C_VEL
LIN {X 0,Y 268.129,Z 548.487,A -85,B 0,C 180,E1 -17724.888,E2 -17724.888} C_VEL
LIN {X 0,Y 268.149,Z 550.036,A -85,B 0,C 180,E1 -17726.995,E2 -17726.995} C_VEL
LIN {X 0,Y 268.184,Z 550.715,A -85,B 0,C 180,E1 -17728.498,E2 -17728.498} C_VEL
LIN {X 0,Y 268.2,Z 551.035,A -85,B 0,C 180,E1 -17730,E2 -17730} C_VEL
LIN {X 0,Y 268.184,Z 550.995,A -85,B 0,C 180,E1 -17731.502,E2 -17731.502} C_VEL
LIN {X 0,Y 268.13,Z 549.84,A -85,B 0,C 180,E1 -17734.51,E2 -17734.51} C_VEL
LIN {X 0,Y 268.217,Z 548.726,A -85,B 0,C 180,E1 -17736.016,E2 -17736.016} C_VEL
LIN {X 0,Y 268.601,Z 545.345,A -85,B 0,C 180,E1 -17739.032,E2 -17739.032} C_VEL
LIN {X 0,Y 269.337,Z 540.367,A -85,B 0,C 180,E1 -17742.049,E2 -17742.049} C_VEL
LIN {X 0,Y 270.413,Z 535.524,A -85,B 0,C 180,E1 -17744.294,E2 -17744.294} C_VEL
LIN {X 0,Y 271.741,Z 529.593,A -85,B 0,C 180,E1 -17746.528,E2 -17746.528} C_VEL
LIN {X 0,Y 273.26,Z 522.389,A -85,B 0,C 180,E1 -17748.753,E2 -17748.753} C_VEL
LIN {X 0,Y 275.286,Z 513.664,A -85,B 0,C 180,E1 -17750.941,E2 -17750.941} C_VEL
LIN {X 0,Y 277.697,Z 503.027,A -85,B 0,C 180,E1 -17753.096,E2 -17753.096} C_VEL
LIN {X 0,Y 280.082,Z 492.238,A -85,B 0,C 180,E1 -17754.853,E2 -17754.853} C_VEL
LIN {X 0,Y 282.188,Z 480.873,A -85,B 0,C 180,E1 -17756.365,E2 -17756.365} C_VEL
LIN {X 0,Y 284.175,Z 468.963,A -85,B 0,C 180,E1 -17757.626,E2 -17757.626} C_VEL
LIN {X 0,Y 286.111,Z 455.514,A -85,B 0,C 180,E1 -17758.72,E2 -17758.72} C_VEL
LIN {X 0,Y 287.589,Z 442.105,A -85,B 0,C 180,E1 -17759.509,E2 -17759.509} C_VEL
LIN {X 0,Y 288.609,Z 428.455,A -85,B 0,C 180,E1 -17760.047,E2 -17760.047} C_VEL
LIN {X 0,Y 292.025,Z 338.976,A -85,B 0,C 180,E1 -17762.303,E2 -17762.303} C_VEL
LIN {X 0,Y 290.359,Z 327.084,A -85,B 0,C 180,E1 -17762.862,E2 -17762.862} C_VEL
LIN {X 0,Y 281.842,Z 308.611,A -85,B 0,C 180,E1 -17764.547,E2 -17764.547} C_VEL
LIN {X 0,Y 278.011,Z 300.899,A -85,B 0,C 180,E1 -17765.388,E2 -17765.388} C_VEL
LIN {X 0,Y 274.913,Z 289.511,A -85,B 0,C 180,E1 -17769.348,E2 -17769.348} C_VEL
LIN {X 0,Y 271.956,Z 279.826,A -85,B 0,C 180,E1 -17773.084,E2 -17773.084} C_VEL
LIN {X 0,Y 270.196,Z 274.531,A -85,B 0,C 180,E1 -17775.389,E2 -17775.389} C_VEL
LIN {X 0,Y 270.173,Z 274.435,A -85,B 0,C 180,E1 -17779.434,E2 -17779.434} C_VEL
LIN {X 0,Y 270.217,Z 274.424,A -85,B 0,C 180,E1 -17783.259,E2 -17783.259} C_VEL
LIN {X 0,Y 270.199,Z 274.454,A -85,B 0,C 180,E1 -17786.892,E2 -17786.892} C_VEL
LIN {X 0,Y 270.193,Z 274.417,A -85,B 0,C 180,E1 -17790.383,E2 -17790.383} C_VEL
LIN {X 0,Y 270.26,Z 274.448,A -85,B 0,C 180,E1 -17793.764,E2 -17793.764} C_VEL
LIN {X 0,Y 270.229,Z 274.449,A -85,B 0,C 180,E1 -17797.039,E2 -17797.039} C_VEL
LIN {X 0,Y 270.298,Z 274.432,A -85,B 0,C 180,E1 -17800.245,E2 -17800.245} C_VEL
LIN {X 0,Y 270.399,Z 274.423,A -85,B 0,C 180,E1 -17804.936,E2 -17804.936} C_VEL
LIN {X 0,Y 270.437,Z 274.417,A -85,B 0,C 180,E1 -17809.519,E2 -17809.519} C_VEL
LIN {X 0,Y 270.603,Z 274.388,A -85,B 0,C 180,E1 -17812.539,E2 -17812.539} C_VEL
LIN {X 0,Y 270.783,Z 274.372,A -85,B 0,C 180,E1 -17818.513,E2 -17818.513} C_VEL
LIN {X 0,Y 270.783,Z 274.369,A -85,B 0,C 180,E1 -17821.488,E2 -17821.488} C_VEL
LIN {X 0,Y 270.607,Z 274.39,A -85,B 0,C 180,E1 -17827.462,E2 -17827.462} C_VEL
LIN {X 0,Y 270.438,Z 274.416,A -85,B 0,C 180,E1 -17830.482,E2 -17830.482} C_VEL
LIN {X 0,Y 270.393,Z 274.42,A -85,B 0,C 180,E1 -17835.066,E2 -17835.066} C_VEL
LIN {X 0,Y 270.3,Z 274.43,A -85,B 0,C 180,E1 -17839.756,E2 -17839.756} C_VEL
LIN {X 0,Y 270.272,Z 274.438,A -85,B 0,C 180,E1 -17844.586,E2 -17844.586} C_VEL
LIN {X 0,Y 270.268,Z 274.417,A -85,B 0,C 180,E1 -17847.91,E2 -17847.91} C_VEL
LIN {X 0,Y 270.183,Z 274.448,A -85,B 0,C 180,E1 -17851.349,E2 -17851.349} C_VEL
LIN {X 0,Y 270.214,Z 274.424,A -85,B 0,C 180,E1 -17854.905,E2 -17854.905} C_VEL
LIN {X 0,Y 270.222,Z 274.437,A -85,B 0,C 180,E1 -17858.718,E2 -17858.718} C_VEL
LIN {X 0,Y 270.196,Z 274.646,A -85,B 0,C 180,E1 -17862.554,E2 -17862.554} C_VEL
LIN {X 0,Y 273.157,Z 284.132,A -85,B 0,C 180,E1 -17866.623,E2 -17866.623} C_VEL
LIN {X 0,Y 275.544,Z 292.585,A -85,B 0,C 180,E1 -17869.924,E2 -17869.924} C_VEL
LIN {X 0,Y 278.007,Z 302.312,A -85,B 0,C 180,E1 -17873.435,E2 -17873.435} C_VEL
LIN {X 0,Y 279.594,Z 309.946,A -85,B 0,C 180,E1 -17875.923,E2 -17875.923} C_VEL
LIN {X 0,Y 284.395,Z 320.582,A -85,B 0,C 180,E1 -17876.927,E2 -17876.927} C_VEL
LIN {X 0,Y 289.212,Z 346.619,A -85,B 0,C 180,E1 -17878.269,E2 -17878.269} C_VEL
LIN {X 0,Y 291.015,Z 357.609,A -85,B 0,C 180,E1 -17878.789,E2 -17878.789} C_VEL
LIN {X 0,Y 288.665,Z 427.426,A -85,B 0,C 180,E1 -17880.428,E2 -17880.428} C_VEL
LIN {X 0,Y 287.562,Z 440.712,A -85,B 0,C 180,E1 -17880.989,E2 -17880.989} C_VEL
LIN {X 0,Y 286.1,Z 454.291,A -85,B 0,C 180,E1 -17881.879,E2 -17881.879} C_VEL
LIN {X 0,Y 284.38,Z 466.518,A -85,B 0,C 180,E1 -17882.985,E2 -17882.985} C_VEL
LIN {X 0,Y 282.283,Z 478.241,A -85,B 0,C 180,E1 -17884.369,E2 -17884.369} C_VEL
LIN {X 0,Y 279.969,Z 488.767,A -85,B 0,C 180,E1 -17885.926,E2 -17885.926} C_VEL
LIN {X 0,Y 277.724,Z 498.306,A -85,B 0,C 180,E1 -17887.692,E2 -17887.692} C_VEL
LIN {X 0,Y 275.696,Z 506.176,A -85,B 0,C 180,E1 -17889.482,E2 -17889.482} C_VEL
LIN {X 0,Y 273.652,Z 513.967,A -85,B 0,C 180,E1 -17891.663,E2 -17891.663} C_VEL
LIN {X 0,Y 272.304,Z 519.276,A -85,B 0,C 180,E1 -17893.507,E2 -17893.507} C_VEL
LIN {X 0,Y 270.906,Z 524.525,A -85,B 0,C 180,E1 -17895.732,E2 -17895.732} C_VEL
LIN {X 0,Y 269.823,Z 528.673,A -85,B 0,C 180,E1 -17897.973,E2 -17897.973} C_VEL
LIN {X 0,Y 268.936,Z 532.699,A -85,B 0,C 180,E1 -17900.979,E2 -17900.979} C_VEL
LIN {X 0,Y 268.391,Z 535.095,A -85,B 0,C 180,E1 -17903.988,E2 -17903.988} C_VEL
LIN {X 0,Y 268.252,Z 536.023,A -85,B 0,C 180,E1 -17906.996,E2 -17906.996} C_VEL
LIN {X 0,Y 268.211,Z 535.535,A -85,B 0,C 180,E1 -17910,E2 -17910} C_VEL
LIN {X 0,Y 268.491,Z 533.538,A -85,B 0,C 180,E1 -17913.001,E2 -17913.001} C_VEL
LIN {X 0,Y 268.805,Z 531.979,A -85,B 0,C 180,E1 -17914.499,E2 -17914.499} C_VEL
LIN {X 0,Y 269.359,Z 528.897,A -85,B 0,C 180,E1 -17916.743,E2 -17916.743} C_VEL
LIN {X 0,Y 270.114,Z 524.844,A -85,B 0,C 180,E1 -17918.981,E2 -17918.981} C_VEL
LIN {X 0,Y 271.169,Z 519.704,A -85,B 0,C 180,E1 -17921.208,E2 -17921.208} C_VEL
LIN {X 0,Y 272.906,Z 512.106,A -85,B 0,C 180,E1 -17923.781,E2 -17923.781} C_VEL
LIN {X 0,Y 274.754,Z 503.969,A -85,B 0,C 180,E1 -17925.96,E2 -17925.96} C_VEL
LIN {X 0,Y 276.517,Z 495.701,A -85,B 0,C 180,E1 -17927.757,E2 -17927.757} C_VEL
LIN {X 0,Y 278.541,Z 485.645,A -85,B 0,C 180,E1 -17929.531,E2 -17929.531} C_VEL
LIN {X 0,Y 280.498,Z 474.381,A -85,B 0,C 180,E1 -17931.11,E2 -17931.11} C_VEL
LIN {X 0,Y 282.297,Z 463.423,A -85,B 0,C 180,E1 -17932.312,E2 -17932.312} C_VEL
LIN {X 0,Y 283.867,Z 451.381,A -85,B 0,C 180,E1 -17933.336,E2 -17933.336} C_VEL
LIN {X 0,Y 285.024,Z 438.45,A -85,B 0,C 180,E1 -17934.147,E2 -17934.147} C_VEL
LIN {X 0,Y 285.908,Z 425.394,A -85,B 0,C 180,E1 -17934.661,E2 -17934.661} C_VEL
LIN {X 0,Y 287.899,Z 355.519,A -85,B 0,C 180,E1 -17936.316,E2 -17936.316} C_VEL
LIN {X 0,Y 283.497,Z 327.916,A -85,B 0,C 180,E1 -17937.558,E2 -17937.558} C_VEL
LIN {X 0,Y 280.8,Z 314.2,A -85,B 0,C 180,E1 -17938.257,E2 -17938.257} C_VEL
LIN {X 0,Y 279.056,Z 309.829,A -85,B 0,C 180,E1 -17938.665,E2 -17938.665} C_VEL
LIN {X 0,Y 277.033,Z 300.157,A -85,B 0,C 180,E1 -17941.762,E2 -17941.762} C_VEL
LIN {X 0,Y 274.517,Z 289.644,A -85,B 0,C 180,E1 -17945.401,E2 -17945.401} C_VEL
LIN {X 0,Y 272.419,Z 281.966,A -85,B 0,C 180,E1 -17948.254,E2 -17948.254} C_VEL
LIN {X 0,Y 270.177,Z 274.505,A -85,B 0,C 180,E1 -17951.312,E2 -17951.312} C_VEL
LIN {X 0,Y 270.152,Z 274.439,A -85,B 0,C 180,E1 -17955.379,E2 -17955.379} C_VEL
LIN {X 0,Y 270.173,Z 274.432,A -85,B 0,C 180,E1 -17959.433,E2 -17959.433} C_VEL
LIN {X 0,Y 270.253,Z 274.444,A -85,B 0,C 180,E1 -17963.721,E2 -17963.721} C_VEL
LIN {X 0,Y 270.202,Z 274.419,A -85,B 0,C 180,E1 -17966.892,E2 -17966.892} C_VEL
LIN {X 0,Y 270.209,Z 274.445,A -85,B 0,C 180,E1 -17970.93,E2 -17970.93} C_VEL
LIN {X 0,Y 270.263,Z 274.445,A -85,B 0,C 180,E1 -17973.763,E2 -17973.763} C_VEL
LIN {X 0,Y 270.209,Z 274.445,A -85,B 0,C 180,E1 -17977.388,E2 -17977.388} C_VEL
LIN {X 0,Y 269.531,Z 274.535,A -85,B 0,C 180,E1 -17978.633,E2 -17978.633} C_VEL
LIN {X 0,Y 266.755,Z 274.883,A -85,B 0,C 180,E1 -17980.663,E2 -17980.663} C_VEL
LIN {X 0,Y 264.419,Z 275.175,A -85,B 0,C 180,E1 -17982.314,E2 -17982.314} C_VEL
LIN {X 0,Y 263.418,Z 275.294,A -85,B 0,C 180,E1 -17983.59,E2 -17983.59} C_VEL
LIN {X 0,Y 263.336,Z 275.3,A -85,B 0,C 180,E1 -17984.023,E2 -17984.023} C_VEL
LIN {X 0,Y 263.331,Z 275.308,A -85,B 0,C 180,E1 -17987.671,E2 -17987.671} C_VEL
LIN {X 0,Y 263.468,Z 275.279,A -85,B 0,C 180,E1 -17990.79,E2 -17990.79} C_VEL
LIN {X 0,Y 263.505,Z 275.281,A -85,B 0,C 180,E1 -17993.875,E2 -17993.875} C_VEL
LIN {X 0,Y 263.747,Z 275.256,A -85,B 0,C 180,E1 -17998.473,E2 -17998.473} C_VEL
LIN {X 0,Y 263.747,Z 275.245,A -85,B 0,C 180,E1 -18001.526,E2 -18001.526} C_VEL
LIN {X 0,Y 263.568,Z 275.275,A -85,B 0,C 180,E1 -18007.661,E2 -18007.661} C_VEL
LIN {X 0,Y 263.369,Z 275.289,A -85,B 0,C 180,E1 -18010.765,E2 -18010.765} C_VEL
LIN {X 0,Y 263.34,Z 275.296,A -85,B 0,C 180,E1 -18015.478,E2 -18015.478} C_VEL
LIN {X 0,Y 263.259,Z 275.306,A -85,B 0,C 180,E1 -18020.307,E2 -18020.307} C_VEL
LIN {X 0,Y 263.204,Z 275.315,A -85,B 0,C 180,E1 -18025.291,E2 -18025.291} C_VEL
LIN {X 0,Y 263.162,Z 275.306,A -85,B 0,C 180,E1 -18028.731,E2 -18028.731} C_VEL
LIN {X 0,Y 263.129,Z 275.314,A -85,B 0,C 180,E1 -18032.288,E2 -18032.288} C_VEL
LIN {X 0,Y 263.159,Z 275.306,A -85,B 0,C 180,E1 -18035.982,E2 -18035.982} C_VEL
LIN {X 0,Y 263.103,Z 275.34,A -85,B 0,C 180,E1 -18039.873,E2 -18039.873} C_VEL
LIN {X 0,Y 263.125,Z 275.33,A -85,B 0,C 180,E1 -18043.983,E2 -18043.983} C_VEL
LIN {X 0,Y 263.135,Z 275.51,A -85,B 0,C 180,E1 -18045.924,E2 -18045.924} C_VEL
LIN {X 0,Y 265.881,Z 284.379,A -85,B 0,C 180,E1 -18049.458,E2 -18049.458} C_VEL
LIN {X 0,Y 268.704,Z 294.186,A -85,B 0,C 180,E1 -18053.019,E2 -18053.019} C_VEL
LIN {X 0,Y 270.409,Z 301.037,A -85,B 0,C 180,E1 -18055.286,E2 -18055.286} C_VEL
LIN {X 0,Y 277.563,Z 316.497,A -85,B 0,C 180,E1 -18056.735,E2 -18056.735} C_VEL
LIN {X 0,Y 281.227,Z 325.108,A -85,B 0,C 180,E1 -18057.443,E2 -18057.443} C_VEL
LIN {X 0,Y 282.813,Z 338.854,A -85,B 0,C 180,E1 -18058.041,E2 -18058.041} C_VEL
LIN {X 0,Y 279.422,Z 430.445,A -85,B 0,C 180,E1 -18060.423,E2 -18060.423} C_VEL
LIN {X 0,Y 278.233,Z 444.874,A -85,B 0,C 180,E1 -18061.062,E2 -18061.062} C_VEL
LIN {X 0,Y 276.734,Z 458.66,A -85,B 0,C 180,E1 -18061.977,E2 -18061.977} C_VEL
LIN {X 0,Y 275.085,Z 470.576,A -85,B 0,C 180,E1 -18063.034,E2 -18063.034} C_VEL
LIN {X 0,Y 273.045,Z 483.442,A -85,B 0,C 180,E1 -18064.502,E2 -18064.502} C_VEL
LIN {X 0,Y 270.958,Z 494.569,A -85,B 0,C 180,E1 -18066.092,E2 -18066.092} C_VEL
LIN {X 0,Y 268.907,Z 504.004,A -85,B 0,C 180,E1 -18067.731,E2 -18067.731} C_VEL
LIN {X 0,Y 267.135,Z 512.858,A -85,B 0,C 180,E1 -18069.599,E2 -18069.599} C_VEL
LIN {X 0,Y 265.301,Z 521.738,A -85,B 0,C 180,E1 -18071.865,E2 -18071.865} C_VEL
LIN {X 0,Y 264.006,Z 529.065,A -85,B 0,C 180,E1 -18074.166,E2 -18074.166} C_VEL
LIN {X 0,Y 262.607,Z 536.014,A -85,B 0,C 180,E1 -18076.852,E2 -18076.852} C_VEL
LIN {X 0,Y 261.821,Z 540.742,A -85,B 0,C 180,E1 -18079.17,E2 -18079.17} C_VEL
LIN {X 0,Y 261.383,Z 544.496,A -85,B 0,C 180,E1 -18081.496,E2 -18081.496} C_VEL
LIN {X 0,Y 261.135,Z 547.364,A -85,B 0,C 180,E1 -18083.82,E2 -18083.82} C_VEL
LIN {X 0,Y 261.043,Z 549.823,A -85,B 0,C 180,E1 -18086.914,E2 -18086.914} C_VEL
LIN {X 0,Y 261.111,Z 550.509,A -85,B 0,C 180,E1 -18088.458,E2 -18088.458} C_VEL
LIN {X 0,Y 261.126,Z 550.834,A -85,B 0,C 180,E1 -18090,E2 -18090} C_VEL
LIN {X 0,Y 261.111,Z 550.799,A -85,B 0,C 180,E1 -18091.542,E2 -18091.542} C_VEL
LIN {X 0,Y 261.045,Z 549.653,A -85,B 0,C 180,E1 -18094.633,E2 -18094.633} C_VEL
LIN {X 0,Y 261.28,Z 547.057,A -85,B 0,C 180,E1 -18097.729,E2 -18097.729} C_VEL
LIN {X 0,Y 261.88,Z 542.894,A -85,B 0,C 180,E1 -18100.828,E2 -18100.828} C_VEL
LIN {X 0,Y 262.716,Z 538.735,A -85,B 0,C 180,E1 -18103.143,E2 -18103.143} C_VEL
LIN {X 0,Y 263.862,Z 533.522,A -85,B 0,C 180,E1 -18105.447,E2 -18105.447} C_VEL
LIN {X 0,Y 265.613,Z 526.103,A -85,B 0,C 180,E1 -18108.085,E2 -18108.085} C_VEL
LIN {X 0,Y 267.52,Z 518.098,A -85,B 0,C 180,E1 -18110.37,E2 -18110.37} C_VEL
LIN {X 0,Y 269.824,Z 508.481,A -85,B 0,C 180,E1 -18112.593,E2 -18112.593} C_VEL
LIN {X 0,Y 272.381,Z 497.761,A -85,B 0,C 180,E1 -18114.586,E2 -18114.586} C_VEL
LIN {X 0,Y 274.759,Z 486.381,A -85,B 0,C 180,E1 -18116.3,E2 -18116.3} C_VEL
LIN {X 0,Y 277.056,Z 474.039,A -85,B 0,C 180,E1 -18117.782,E2 -18117.782} C_VEL
LIN {X 0,Y 279.091,Z 461.004,A -85,B 0,C 180,E1 -18118.996,E2 -18118.996} C_VEL
LIN {X 0,Y 280.898,Z 447.359,A -85,B 0,C 180,E1 -18119.922,E2 -18119.922} C_VEL
LIN {X 0,Y 282.12,Z 434.231,A -85,B 0,C 180,E1 -18120.553,E2 -18120.553} C_VEL
LIN {X 0,Y 283.051,Z 416.878,A -85,B 0,C 180,E1 -18121.063,E2 -18121.063} C_VEL
LIN {X 0,Y 285.943,Z 338.962,A -85,B 0,C 180,E1 -18123.065,E2 -18123.065} C_VEL
LIN {X 0,Y 284.545,Z 329.641,A -85,B 0,C 180,E1 -18123.531,E2 -18123.531} C_VEL
LIN {X 0,Y 276.596,Z 312.392,A -85,B 0,C 180,E1 -18125.166,E2 -18125.166} C_VEL
LIN {X 0,Y 270.918,Z 301.202,A -85,B 0,C 180,E1 -18126.412,E2 -18126.412} C_VEL
LIN {X 0,Y 267.855,Z 290.059,A -85,B 0,C 180,E1 -18130.457,E2 -18130.457} C_VEL
LIN {X 0,Y 264.932,Z 280.704,A -85,B 0,C 180,E1 -18134.255,E2 -18134.255} C_VEL
LIN {X 0,Y 263.157,Z 275.387,A -85,B 0,C 180,E1 -18136.684,E2 -18136.684} C_VEL
LIN {X 0,Y 263.133,Z 275.329,A -85,B 0,C 180,E1 -18140.764,E2 -18140.764} C_VEL
LIN {X 0,Y 263.161,Z 275.3,A -85,B 0,C 180,E1 -18144.018,E2 -18144.018} C_VEL
LIN {X 0,Y 263.129,Z 275.327,A -85,B 0,C 180,E1 -18147.712,E2 -18147.712} C_VEL
LIN {X 0,Y 263.193,Z 275.3,A -85,B 0,C 180,E1 -18151.785,E2 -18151.785} C_VEL
LIN {X 0,Y 263.222,Z 275.313,A -85,B 0,C 180,E1 -18155.2,E2 -18155.2} C_VEL
LIN {X 0,Y 263.26,Z 275.306,A -85,B 0,C 180,E1 -18159.694,E2 -18159.694} C_VEL
LIN {X 0,Y 263.347,Z 275.297,A -85,B 0,C 180,E1 -18164.522,E2 -18164.522} C_VEL
LIN {X 0,Y 263.37,Z 275.295,A -85,B 0,C 180,E1 -18169.235,E2 -18169.235} C_VEL
LIN {X 0,Y 263.565,Z 275.265,A -85,B 0,C 180,E1 -18172.339,E2 -18172.339} C_VEL
LIN {X 0,Y 263.747,Z 275.247,A -85,B 0,C 180,E1 -18178.474,E2 -18178.474} C_VEL
LIN {X 0,Y 263.748,Z 275.245,A -85,B 0,C 180,E1 -18181.527,E2 -18181.527} C_VEL
LIN {X 0,Y 263.569,Z 275.267,A -85,B 0,C 180,E1 -18187.662,E2 -18187.662} C_VEL
LIN {X 0,Y 263.371,Z 275.293,A -85,B 0,C 180,E1 -18190.766,E2 -18190.766} C_VEL
LIN {X 0,Y 263.342,Z 275.295,A -85,B 0,C 180,E1 -18195.479,E2 -18195.479} C_VEL
LIN {X 0,Y 263.262,Z 275.306,A -85,B 0,C 180,E1 -18200.307,E2 -18200.307} C_VEL
LIN {X 0,Y 263.207,Z 275.324,A -85,B 0,C 180,E1 -18205.292,E2 -18205.292} C_VEL
LIN {X 0,Y 263.164,Z 275.295,A -85,B 0,C 180,E1 -18208.732,E2 -18208.732} C_VEL
LIN {X 0,Y 263.132,Z 275.336,A -85,B 0,C 180,E1 -18212.289,E2 -18212.289} C_VEL
LIN {X 0,Y 263.187,Z 275.303,A -85,B 0,C 180,E1 -18215.979,E2 -18215.979} C_VEL
LIN {X 0,Y 263.114,Z 275.313,A -85,B 0,C 180,E1 -18219.872,E2 -18219.872} C_VEL
LIN {X 0,Y 263.164,Z 275.516,A -85,B 0,C 180,E1 -18221.276,E2 -18221.276} C_VEL
LIN {X 0,Y 266.098,Z 284.851,A -85,B 0,C 180,E1 -18225.489,E2 -18225.489} C_VEL
LIN {X 0,Y 268.786,Z 294.234,A -85,B 0,C 180,E1 -18229.313,E2 -18229.313} C_VEL
LIN {X 0,Y 271.327,Z 304.374,A -85,B 0,C 180,E1 -18233.088,E2 -18233.088} C_VEL
LIN {X 0,Y 272.521,Z 309.882,A -85,B 0,C 180,E1 -18234.906,E2 -18234.906} C_VEL
LIN {X 0,Y 278.725,Z 323.222,A -85,B 0,C 180,E1 -18236.234,E2 -18236.234} C_VEL
LIN {X 0,Y 283.334,Z 348.589,A -85,B 0,C 180,E1 -18237.58,E2 -18237.58} C_VEL
LIN {X 0,Y 284.915,Z 359.383,A -85,B 0,C 180,E1 -18238.085,E2 -18238.085} C_VEL
LIN {X 0,Y 282.523,Z 427.719,A -85,B 0,C 180,E1 -18239.726,E2 -18239.726} C_VEL
LIN {X 0,Y 281.3,Z 441.588,A -85,B 0,C 180,E1 -18240.331,E2 -18240.331} C_VEL
LIN {X 0,Y 279.849,Z 454.387,A -85,B 0,C 180,E1 -18241.193,E2 -18241.193} C_VEL
LIN {X 0,Y 278.07,Z 466.613,A -85,B 0,C 180,E1 -18242.32,E2 -18242.32} C_VEL
LIN {X 0,Y 275.903,Z 478.34,A -85,B 0,C 180,E1 -18243.731,E2 -18243.731} C_VEL
LIN {X 0,Y 273.508,Z 488.872,A -85,B 0,C 180,E1 -18245.32,E2 -18245.32} C_VEL
LIN {X 0,Y 271.128,Z 498.418,A -85,B 0,C 180,E1 -18247.119,E2 -18247.119} C_VEL
LIN {X 0,Y 269.033,Z 506.296,A -85,B 0,C 180,E1 -18248.95,E2 -18248.95} C_VEL
LIN {X 0,Y 266.906,Z 514.096,A -85,B 0,C 180,E1 -18251.183,E2 -18251.183} C_VEL
LIN {X 0,Y 265.001,Z 521.303,A -85,B 0,C 180,E1 -18253.831,E2 -18253.831} C_VEL
LIN {X 0,Y 263.521,Z 526.187,A -85,B 0,C 180,E1 -18256.112,E2 -18256.112} C_VEL
LIN {X 0,Y 262.571,Z 530.016,A -85,B 0,C 180,E1 -18258.42,E2 -18258.42} C_VEL
LIN {X 0,Y 261.899,Z 532.868,A -85,B 0,C 180,E1 -18260.735,E2 -18260.735} C_VEL
LIN {X 0,Y 261.316,Z 535.279,A -85,B 0,C 180,E1 -18263.824,E2 -18263.824} C_VEL
LIN {X 0,Y 261.165,Z 536.219,A -85,B 0,C 180,E1 -18266.915,E2 -18266.915} C_VEL
LIN {X 0,Y 261.137,Z 535.745,A -85,B 0,C 180,E1 -18270,E2 -18270} C_VEL
LIN {X 0,Y 261.43,Z 533.764,A -85,B 0,C 180,E1 -18273.082,E2 -18273.082} C_VEL
LIN {X 0,Y 262.094,Z 530.278,A -85,B 0,C 180,E1 -18276.157,E2 -18276.157} C_VEL
LIN {X 0,Y 262.811,Z 526.565,A -85,B 0,C 180,E1 -18278.457,E2 -18278.457} C_VEL
LIN {X 0,Y 263.799,Z 521.813,A -85,B 0,C 180,E1 -18280.748,E2 -18280.748} C_VEL
LIN {X 0,Y 265.44,Z 514.791,A -85,B 0,C 180,E1 -18283.395,E2 -18283.395} C_VEL
LIN {X 0,Y 267.269,Z 507.227,A -85,B 0,C 180,E1 -18285.636,E2 -18285.636} C_VEL
LIN {X 0,Y 269.425,Z 497.831,A -85,B 0,C 180,E1 -18287.848,E2 -18287.848} C_VEL
LIN {X 0,Y 271.382,Z 488.228,A -85,B 0,C 180,E1 -18289.673,E2 -18289.673} C_VEL
LIN {X 0,Y 273.491,Z 477.615,A -85,B 0,C 180,E1 -18291.283,E2 -18291.283} C_VEL
LIN {X 0,Y 275.552,Z 465.799,A -85,B 0,C 180,E1 -18292.691,E2 -18292.691} C_VEL
LIN {X 0,Y 277.258,Z 453.287,A -85,B 0,C 180,E1 -18293.827,E2 -18293.827} C_VEL
LIN {X 0,Y 278.579,Z 439.886,A -85,B 0,C 180,E1 -18294.717,E2 -18294.717} C_VEL
LIN {X 0,Y 279.578,Z 426.15,A -85,B 0,C 180,E1 -18295.299,E2 -18295.299} C_VEL
LIN {X 0,Y 281.679,Z 356.542,A -85,B 0,C 180,E1 -18296.983,E2 -18296.983} C_VEL
LIN {X 0,Y 277.509,Z 329.913,A -85,B 0,C 180,E1 -18298.216,E2 -18298.216} C_VEL
LIN {X 0,Y 275.003,Z 316.973,A -85,B 0,C 180,E1 -18298.895,E2 -18298.895} C_VEL
LIN {X 0,Y 271.92,Z 309.749,A -85,B 0,C 180,E1 -18299.567,E2 -18299.567} C_VEL
LIN {X 0,Y 269.881,Z 300.28,A -85,B 0,C 180,E1 -18302.707,E2 -18302.707} C_VEL
LIN {X 0,Y 267.51,Z 290.493,A -85,B 0,C 180,E1 -18306.235,E2 -18306.235} C_VEL
LIN {X 0,Y 265.729,Z 284.038,A -85,B 0,C 180,E1 -18308.72,E2 -18308.72} C_VEL
LIN {X 0,Y 263.146,Z 275.396,A -85,B 0,C 180,E1 -18312.379,E2 -18312.379} C_VEL
LIN {X 0,Y 263.105,Z 275.321,A -85,B 0,C 180,E1 -18316.154,E2 -18316.154} C_VEL
LIN {X 0,Y 263.113,Z 275.308,A -85,B 0,C 180,E1 -18320.128,E2 -18320.128} C_VEL
LIN {X 0,Y 263.186,Z 275.316,A -85,B 0,C 180,E1 -18324.021,E2 -18324.021} C_VEL
LIN {X 0,Y 263.132,Z 275.307,A -85,B 0,C 180,E1 -18327.711,E2 -18327.711} C_VEL
LIN {X 0,Y 263.197,Z 275.315,A -85,B 0,C 180,E1 -18331.783,E2 -18331.783} C_VEL
LIN {X 0,Y 263.224,Z 275.311,A -85,B 0,C 180,E1 -18335.199,E2 -18335.199} C_VEL
LIN {X 0,Y 263.261,Z 275.307,A -85,B 0,C 180,E1 -18339.693,E2 -18339.693} C_VEL
LIN {X 0,Y 263.336,Z 275.3,A -85,B 0,C 180,E1 -18344.023,E2 -18344.023} C_VEL
LIN {X 0,Y 262.678,Z 275.379,A -85,B 0,C 180,E1 -18345.298,E2 -18345.298} C_VEL
LIN {X 0,Y 259.877,Z 275.739,A -85,B 0,C 180,E1 -18347.379,E2 -18347.379} C_VEL
LIN {X 0,Y 257.51,Z 276.026,A -85,B 0,C 180,E1 -18349.071,E2 -18349.071} C_VEL
LIN {X 0,Y 256.507,Z 276.144,A -85,B 0,C 180,E1 -18350.381,E2 -18350.381} C_VEL
LIN {X 0,Y 256.432,Z 276.154,A -85,B 0,C 180,E1 -18350.825,E2 -18350.825} C_VEL
LIN {X 0,Y 256.477,Z 276.159,A -85,B 0,C 180,E1 -18353.707,E2 -18353.707} C_VEL
LIN {X 0,Y 256.71,Z 276.133,A -85,B 0,C 180,E1 -18358.431,E2 -18358.431} C_VEL
LIN {X 0,Y 256.71,Z 276.121,A -85,B 0,C 180,E1 -18361.568,E2 -18361.568} C_VEL
LIN {X 0,Y 256.535,Z 276.152,A -85,B 0,C 180,E1 -18367.873,E2 -18367.873} C_VEL
LIN {X 0,Y 256.305,Z 276.168,A -85,B 0,C 180,E1 -18371.066,E2 -18371.066} C_VEL
LIN {X 0,Y 256.29,Z 276.172,A -85,B 0,C 180,E1 -18375.915,E2 -18375.915} C_VEL
LIN {X 0,Y 256.162,Z 276.19,A -85,B 0,C 180,E1 -18380.895,E2 -18380.895} C_VEL
LIN {X 0,Y 256.184,Z 276.188,A -85,B 0,C 180,E1 -18385.138,E2 -18385.138} C_VEL
LIN {X 0,Y 256.1,Z 276.174,A -85,B 0,C 180,E1 -18389.601,E2 -18389.601} C_VEL
LIN {X 0,Y 256.072,Z 276.212,A -85,B 0,C 180,E1 -18393.292,E2 -18393.292} C_VEL
LIN {X 0,Y 256.11,Z 276.181,A -85,B 0,C 180,E1 -18397.271,E2 -18397.271} C_VEL
LIN {X 0,Y 256.051,Z 276.198,A -85,B 0,C 180,E1 -18401.204,E2 -18401.204} C_VEL
LIN {X 0,Y 256.117,Z 276.432,A -85,B 0,C 180,E1 -18404.775,E2 -18404.775} C_VEL
LIN {X 0,Y 258.786,Z 284.875,A -85,B 0,C 180,E1 -18408.316,E2 -18408.316} C_VEL
LIN {X 0,Y 261.437,Z 294.052,A -85,B 0,C 180,E1 -18411.809,E2 -18411.809} C_VEL
LIN {X 0,Y 263.26,Z 301.214,A -85,B 0,C 180,E1 -18414.298,E2 -18414.298} C_VEL
LIN {X 0,Y 270.404,Z 316.271,A -85,B 0,C 180,E1 -18415.81,E2 -18415.81} C_VEL
LIN {X 0,Y 275.296,Z 327.683,A -85,B 0,C 180,E1 -18416.798,E2 -18416.798} C_VEL
LIN {X 0,Y 276.654,Z 339.018,A -85,B 0,C 180,E1 -18417.314,E2 -18417.314} C_VEL
LIN {X 0,Y 273.162,Z 430.176,A -85,B 0,C 180,E1 -18419.728,E2 -18419.728} C_VEL
LIN {X 0,Y 272.058,Z 443.939,A -85,B 0,C 180,E1 -18420.34,E2 -18420.34} C_VEL
LIN {X 0,Y 270.599,Z 456.808,A -85,B 0,C 180,E1 -18421.178,E2 -18421.178} C_VEL
LIN {X 0,Y 268.73,Z 469.99,A -85,B 0,C 180,E1 -18422.342,E2 -18422.342} C_VEL
LIN {X 0,Y 266.685,Z 482.447,A -85,B 0,C 180,E1 -18423.776,E2 -18423.776} C_VEL
LIN {X 0,Y 264.457,Z 494.14,A -85,B 0,C 180,E1 -18425.466,E2 -18425.466} C_VEL
LIN {X 0,Y 261.923,Z 505.546,A -85,B 0,C 180,E1 -18427.521,E2 -18427.521} C_VEL
LIN {X 0,Y 259.745,Z 515.672,A -85,B 0,C 180,E1 -18429.82,E2 -18429.82} C_VEL
LIN {X 0,Y 257.98,Z 524.016,A -85,B 0,C 180,E1 -18432.153,E2 -18432.153} C_VEL
LIN {X 0,Y 256.609,Z 530.914,A -85,B 0,C 180,E1 -18434.513,E2 -18434.513} C_VEL
LIN {X 0,Y 255.278,Z 537.417,A -85,B 0,C 180,E1 -18437.277,E2 -18437.277} C_VEL
LIN {X 0,Y 254.605,Z 541.851,A -85,B 0,C 180,E1 -18439.664,E2 -18439.664} C_VEL
LIN {X 0,Y 254.217,Z 545.341,A -85,B 0,C 180,E1 -18442.055,E2 -18442.055} C_VEL
LIN {X 0,Y 253.927,Z 548.557,A -85,B 0,C 180,E1 -18445.237,E2 -18445.237} C_VEL
LIN {X 0,Y 254.016,Z 550.303,A -85,B 0,C 180,E1 -18448.415,E2 -18448.415} C_VEL
LIN {X 0,Y 254.053,Z 550.633,A -85,B 0,C 180,E1 -18450,E2 -18450} C_VEL
LIN {X 0,Y 254.016,Z 550.603,A -85,B 0,C 180,E1 -18451.585,E2 -18451.585} C_VEL
LIN {X 0,Y 253.972,Z 549.467,A -85,B 0,C 180,E1 -18454.762,E2 -18454.762} C_VEL
LIN {X 0,Y 254.219,Z 546.882,A -85,B 0,C 180,E1 -18457.945,E2 -18457.945} C_VEL
LIN {X 0,Y 254.875,Z 542.728,A -85,B 0,C 180,E1 -18461.129,E2 -18461.129} C_VEL
LIN {X 0,Y 255.771,Z 538.576,A -85,B 0,C 180,E1 -18463.507,E2 -18463.507} C_VEL
LIN {X 0,Y 256.991,Z 533.368,A -85,B 0,C 180,E1 -18465.871,E2 -18465.871} C_VEL
LIN {X 0,Y 258.838,Z 525.874,A -85,B 0,C 180,E1 -18468.604,E2 -18468.604} C_VEL
LIN {X 0,Y 260.822,Z 517.959,A -85,B 0,C 180,E1 -18470.918,E2 -18470.918} C_VEL
LIN {X 0,Y 263.231,Z 508.346,A -85,B 0,C 180,E1 -18473.191,E2 -18473.191} C_VEL
LIN {X 0,Y 265.906,Z 497.63,A -85,B 0,C 180,E1 -18475.226,E2 -18475.226} C_VEL
LIN {X 0,Y 268.216,Z 487.1,A -85,B 0,C 180,E1 -18476.855,E2 -18476.855} C_VEL
LIN {X 0,Y 270.485,Z 475.491,A -85,B 0,C 180,E1 -18478.306,E2 -18478.306} C_VEL
LIN {X 0,Y 272.742,Z 461.906,A -85,B 0,C 180,E1 -18479.631,E2 -18479.631} C_VEL
LIN {X 0,Y 274.684,Z 447.937,A -85,B 0,C 180,E1 -18480.618,E2 -18480.618} C_VEL
LIN {X 0,Y 276.034,Z 433.996,A -85,B 0,C 180,E1 -18481.302,E2 -18481.302} C_VEL
LIN {X 0,Y 276.991,Z 416.525,A -85,B 0,C 180,E1 -18481.821,E2 -18481.821} C_VEL
LIN {X 0,Y 279.967,Z 339.894,A -85,B 0,C 180,E1 -18483.823,E2 -18483.823} C_VEL
LIN {X 0,Y 278.796,Z 332.268,A -85,B 0,C 180,E1 -18484.222,E2 -18484.222} C_VEL
LIN {X 0,Y 271.407,Z 316.208,A -85,B 0,C 180,E1 -18485.804,E2 -18485.804} C_VEL
LIN {X 0,Y 265.438,Z 304.639,A -85,B 0,C 180,E1 -18487.118,E2 -18487.118} C_VEL
LIN {X 0,Y 263.728,Z 301.278,A -85,B 0,C 180,E1 -18487.565,E2 -18487.565} C_VEL
LIN {X 0,Y 261.173,Z 291.95,A -85,B 0,C 180,E1 -18491.109,E2 -18491.109} C_VEL
LIN {X 0,Y 258.638,Z 283.882,A -85,B 0,C 180,E1 -18494.497,E2 -18494.497} C_VEL
LIN {X 0,Y 256.104,Z 276.243,A -85,B 0,C 180,E1 -18498.119,E2 -18498.119} C_VEL
LIN {X 0,Y 256.129,Z 276.181,A -85,B 0,C 180,E1 -18502.868,E2 -18502.868} C_VEL
LIN {X 0,Y 256.064,Z 276.215,A -85,B 0,C 180,E1 -18506.707,E2 -18506.707} C_VEL
LIN {X 0,Y 256.1,Z 276.171,A -85,B 0,C 180,E1 -18510.399,E2 -18510.399} C_VEL
LIN {X 0,Y 256.185,Z 276.191,A -85,B 0,C 180,E1 -18514.862,E2 -18514.862} C_VEL
LIN {X 0,Y 256.163,Z 276.191,A -85,B 0,C 180,E1 -18519.105,E2 -18519.105} C_VEL
LIN {X 0,Y 256.296,Z 276.172,A -85,B 0,C 180,E1 -18524.085,E2 -18524.085} C_VEL
LIN {X 0,Y 256.306,Z 276.172,A -85,B 0,C 180,E1 -18528.934,E2 -18528.934} C_VEL
LIN {X 0,Y 256.534,Z 276.142,A -85,B 0,C 180,E1 -18532.127,E2 -18532.127} C_VEL
LIN {X 0,Y 256.71,Z 276.123,A -85,B 0,C 180,E1 -18538.432,E2 -18538.432} C_VEL
LIN {X 0,Y 256.711,Z 276.121,A -85,B 0,C 180,E1 -18541.569,E2 -18541.569} C_VEL
LIN {X 0,Y 256.537,Z 276.145,A -85,B 0,C 180,E1 -18547.874,E2 -18547.874} C_VEL
LIN {X 0,Y 256.306,Z 276.171,A -85,B 0,C 180,E1 -18551.067,E2 -18551.067} C_VEL
LIN {X 0,Y 256.292,Z 276.173,A -85,B 0,C 180,E1 -18555.916,E2 -18555.916} C_VEL
LIN {X 0,Y 256.167,Z 276.193,A -85,B 0,C 180,E1 -18560.896,E2 -18560.896} C_VEL
LIN {X 0,Y 256.187,Z 276.197,A -85,B 0,C 180,E1 -18565.139,E2 -18565.139} C_VEL
LIN {X 0,Y 256.102,Z 276.174,A -85,B 0,C 180,E1 -18569.602,E2 -18569.602} C_VEL
LIN {X 0,Y 256.084,Z 276.198,A -85,B 0,C 180,E1 -18573.291,E2 -18573.291} C_VEL
LIN {X 0,Y 256.128,Z 276.201,A -85,B 0,C 180,E1 -18577.276,E2 -18577.276} C_VEL
LIN {X 0,Y 256.111,Z 276.437,A -85,B 0,C 180,E1 -18579.909,E2 -18579.909} C_VEL
LIN {X 0,Y 258.723,Z 284.642,A -85,B 0,C 180,E1 -18583.844,E2 -18583.844} C_VEL
LIN {X 0,Y 261.103,Z 292.492,A -85,B 0,C 180,E1 -18587.274,E2 -18587.274} C_VEL
LIN {X 0,Y 263.333,Z 301.108,A -85,B 0,C 180,E1 -18590.713,E2 -18590.713} C_VEL
LIN {X 0,Y 265.293,Z 309.429,A -85,B 0,C 180,E1 -18593.734,E2 -18593.734} C_VEL
LIN {X 0,Y 268.306,Z 315.914,A -85,B 0,C 180,E1 -18594.488,E2 -18594.488} C_VEL
LIN {X 0,Y 273.193,Z 326.348,A -85,B 0,C 180,E1 -18595.54,E2 -18595.54} C_VEL
LIN {X 0,Y 277.746,Z 352.17,A -85,B 0,C 180,E1 -18596.941,E2 -18596.941} C_VEL
LIN {X 0,Y 278.925,Z 360.084,A -85,B 0,C 180,E1 -18597.328,E2 -18597.328} C_VEL
LIN {X 0,Y 276.421,Z 428.02,A -85,B 0,C 180,E1 -18598.992,E2 -18598.992} C_VEL
LIN {X 0,Y 275.175,Z 441.692,A -85,B 0,C 180,E1 -18599.602,E2 -18599.602} C_VEL
LIN {X 0,Y 273.64,Z 454.483,A -85,B 0,C 180,E1 -18600.476,E2 -18600.476} C_VEL
LIN {X 0,Y 271.831,Z 466.542,A -85,B 0,C 180,E1 -18601.606,E2 -18601.606} C_VEL
LIN {X 0,Y 269.56,Z 478.439,A -85,B 0,C 180,E1 -18603.064,E2 -18603.064} C_VEL
LIN {X 0,Y 267.077,Z 488.976,A -85,B 0,C 180,E1 -18604.684,E2 -18604.684} C_VEL
LIN {X 0,Y 264.581,Z 498.531,A -85,B 0,C 180,E1 -18606.52,E2 -18606.52} C_VEL
LIN {X 0,Y 262.413,Z 506.416,A -85,B 0,C 180,E1 -18608.392,E2 -18608.392} C_VEL
LIN {X 0,Y 260.171,Z 514.225,A -85,B 0,C 180,E1 -18610.676,E2 -18610.676} C_VEL
LIN {X 0,Y 258.63,Z 519.553,A -85,B 0,C 180,E1 -18612.608,E2 -18612.608} C_VEL
LIN {X 0,Y 257.142,Z 524.82,A -85,B 0,C 180,E1 -18614.951,E2 -18614.951} C_VEL
LIN {X 0,Y 255.874,Z 528.989,A -85,B 0,C 180,E1 -18617.307,E2 -18617.307} C_VEL
LIN {X 0,Y 255.326,Z 531.215,A -85,B 0,C 180,E1 -18618.891,E2 -18618.891} C_VEL
LIN {X 0,Y 254.857,Z 533.037,A -85,B 0,C 180,E1 -18620.476,E2 -18620.476} C_VEL
LIN {X 0,Y 254.497,Z 534.45,A -85,B 0,C 180,E1 -18622.064,E2 -18622.064} C_VEL
LIN {X 0,Y 254.099,Z 536.118,A -85,B 0,C 180,E1 -18625.24,E2 -18625.24} C_VEL
LIN {X 0,Y 254.074,Z 536.36,A -85,B 0,C 180,E1 -18628.415,E2 -18628.415} C_VEL
LIN {X 0,Y 254.154,Z 535.162,A -85,B 0,C 180,E1 -18631.584,E2 -18631.584} C_VEL
LIN {X 0,Y 254.668,Z 532.447,A -85,B 0,C 180,E1 -18634.749,E2 -18634.749} C_VEL
LIN {X 0,Y 255.272,Z 529.24,A -85,B 0,C 180,E1 -18637.219,E2 -18637.219} C_VEL
LIN {X 0,Y 256.433,Z 523.805,A -85,B 0,C 180,E1 -18640.261,E2 -18640.261} C_VEL
LIN {X 0,Y 258.017,Z 517.275,A -85,B 0,C 180,E1 -18642.986,E2 -18642.986} C_VEL
LIN {X 0,Y 259.843,Z 510.224,A -85,B 0,C 180,E1 -18645.29,E2 -18645.29} C_VEL
LIN {X 0,Y 261.897,Z 501.538,A -85,B 0,C 180,E1 -18647.571,E2 -18647.571} C_VEL
LIN {X 0,Y 263.865,Z 492.706,A -85,B 0,C 180,E1 -18649.447,E2 -18649.447} C_VEL
LIN {X 0,Y 266.209,Z 481.901,A -85,B 0,C 180,E1 -18651.284,E2 -18651.284} C_VEL
LIN {X 0,Y 268.244,Z 471.128,A -85,B 0,C 180,E1 -18652.733,E2 -18652.733} C_VEL
LIN {X 0,Y 270.147,Z 459.188,A -85,B 0,C 180,E1 -18653.984,E2 -18653.984} C_VEL
LIN {X 0,Y 271.672,Z 446.545,A -85,B 0,C 180,E1 -18654.986,E2 -18654.986} C_VEL
LIN {X 0,Y 272.735,Z 434.437,A -85,B 0,C 180,E1 -18655.669,E2 -18655.669} C_VEL
LIN {X 0,Y 273.506,Z 421.433,A -85,B 0,C 180,E1 -18656.124,E2 -18656.124} C_VEL
LIN {X 0,Y 275.484,Z 357.128,A -85,B 0,C 180,E1 -18657.694,E2 -18657.694} C_VEL
LIN {X 0,Y 270.84,Z 327.761,A -85,B 0,C 180,E1 -18659.116,E2 -18659.116} C_VEL
LIN {X 0,Y 269.229,Z 319.855,A -85,B 0,C 180,E1 -18659.558,E2 -18659.558} C_VEL
LIN {X 0,Y 264.82,Z 309.703,A -85,B 0,C 180,E1 -18660.518,E2 -18660.518} C_VEL
LIN {X 0,Y 262.454,Z 299.005,A -85,B 0,C 180,E1 -18664.217,E2 -18664.217} C_VEL
LIN {X 0,Y 260.096,Z 289.532,A -85,B 0,C 180,E1 -18667.823,E2 -18667.823} C_VEL
LIN {X 0,Y 257.14,Z 279.898,A -85,B 0,C 180,E1 -18671.86,E2 -18671.86} C_VEL
LIN {X 0,Y 256.085,Z 276.258,A -85,B 0,C 180,E1 -18673.591,E2 -18673.591} C_VEL
LIN {X 0,Y 256.069,Z 276.212,A -85,B 0,C 180,E1 -18677.818,E2 -18677.818} C_VEL
LIN {X 0,Y 256.087,Z 276.185,A -85,B 0,C 180,E1 -18680.86,E2 -18680.86} C_VEL
LIN {X 0,Y 256.119,Z 276.181,A -85,B 0,C 180,E1 -18684.812,E2 -18684.812} C_VEL
LIN {X 0,Y 256.091,Z 276.198,A -85,B 0,C 180,E1 -18688.571,E2 -18688.571} C_VEL
LIN {X 0,Y 256.139,Z 276.195,A -85,B 0,C 180,E1 -18692.195,E2 -18692.195} C_VEL
LIN {X 0,Y 256.165,Z 276.189,A -85,B 0,C 180,E1 -18695.698,E2 -18695.698} C_VEL
LIN {X 0,Y 256.164,Z 276.195,A -85,B 0,C 180,E1 -18699.104,E2 -18699.104} C_VEL
LIN {X 0,Y 256.291,Z 276.176,A -85,B 0,C 180,E1 -18704.084,E2 -18704.084} C_VEL
LIN {X 0,Y 256.29,Z 276.186,A -85,B 0,C 180,E1 -18707.327,E2 -18707.327} C_VEL
LIN {X 0,Y 256.432,Z 276.154,A -85,B 0,C 180,E1 -18710.825,E2 -18710.825} C_VEL
LIN {X 0,Y 255.76,Z 276.251,A -85,B 0,C 180,E1 -18712.135,E2 -18712.135} C_VEL
LIN {X 0,Y 252.867,Z 276.601,A -85,B 0,C 180,E1 -18714.27,E2 -18714.27} C_VEL
LIN {X 0,Y 250.485,Z 276.896,A -85,B 0,C 180,E1 -18716.008,E2 -18716.008} C_VEL
LIN {X 0,Y 249.576,Z 277.021,A -85,B 0,C 180,E1 -18717.357,E2 -18717.357} C_VEL
LIN {X 0,Y 249.563,Z 277.018,A -85,B 0,C 180,E1 -18717.813,E2 -18717.813} C_VEL
LIN {X 0,Y 249.723,Z 276.99,A -85,B 0,C 180,E1 -18719.999,E2 -18719.999} C_VEL
LIN {X 0,Y 249.432,Z 277.039,A -85,B 0,C 180,E1 -18723.23,E2 -18723.23} C_VEL
LIN {X 0,Y 249.477,Z 277.032,A -85,B 0,C 180,E1 -18728.097,E2 -18728.097} C_VEL
LIN {X 0,Y 249.248,Z 277.047,A -85,B 0,C 180,E1 -18731.383,E2 -18731.383} C_VEL
LIN {X 0,Y 249.214,Z 277.055,A -85,B 0,C 180,E1 -18736.503,E2 -18736.503} C_VEL
LIN {X 0,Y 249.083,Z 277.076,A -85,B 0,C 180,E1 -18741.518,E2 -18741.518} C_VEL
LIN {X 0,Y 249.127,Z 277.069,A -85,B 0,C 180,E1 -18745.482,E2 -18745.482} C_VEL
LIN {X 0,Y 249.069,Z 277.056,A -85,B 0,C 180,E1 -18748.989,E2 -18748.989} C_VEL
LIN {X 0,Y 249.029,Z 277.071,A -85,B 0,C 180,E1 -18752.426,E2 -18752.426} C_VEL
LIN {X 0,Y 249.053,Z 277.059,A -85,B 0,C 180,E1 -18756.341,E2 -18756.341} C_VEL
LIN {X 0,Y 249.003,Z 277.085,A -85,B 0,C 180,E1 -18760.478,E2 -18760.478} C_VEL
LIN {X 0,Y 249.049,Z 277.263,A -85,B 0,C 180,E1 -18763.474,E2 -18763.474} C_VEL
LIN {X 0,Y 252.399,Z 287.746,A -85,B 0,C 180,E1 -18768.067,E2 -18768.067} C_VEL
LIN {X 0,Y 255.037,Z 297.147,A -85,B 0,C 180,E1 -18771.746,E2 -18771.746} C_VEL
LIN {X 0,Y 256.22,Z 301.453,A -85,B 0,C 180,E1 -18773.269,E2 -18773.269} C_VEL
LIN {X 0,Y 264.563,Z 318.853,A -85,B 0,C 180,E1 -18775.102,E2 -18775.102} C_VEL
LIN {X 0,Y 269.411,Z 330.181,A -85,B 0,C 180,E1 -18776.123,E2 -18776.123} C_VEL
LIN {X 0,Y 270.503,Z 340.859,A -85,B 0,C 180,E1 -18776.603,E2 -18776.603} C_VEL
LIN {X 0,Y 266.862,Z 431.089,A -85,B 0,C 180,E1 -18779.045,E2 -18779.045} C_VEL
LIN {X 0,Y 265.622,Z 445.269,A -85,B 0,C 180,E1 -18779.711,E2 -18779.711} C_VEL
LIN {X 0,Y 264.073,Z 458.351,A -85,B 0,C 180,E1 -18780.615,E2 -18780.615} C_VEL
LIN {X 0,Y 262.14,Z 471.177,A -85,B 0,C 180,E1 -18781.802,E2 -18781.802} C_VEL
LIN {X 0,Y 260.094,Z 483.06,A -85,B 0,C 180,E1 -18783.225,E2 -18783.225} C_VEL
LIN {X 0,Y 257.73,Z 494.888,A -85,B 0,C 180,E1 -18784.998,E2 -18784.998} C_VEL
LIN {X 0,Y 255.316,Z 505.184,A -85,B 0,C 180,E1 -18786.906,E2 -18786.906} C_VEL
LIN {X 0,Y 253.02,Z 515.343,A -85,B 0,C 180,E1 -18789.259,E2 -18789.259} C_VEL
LIN {X 0,Y 251.161,Z 523.714,A -85,B 0,C 180,E1 -18791.652,E2 -18791.652} C_VEL
LIN {X 0,Y 249.743,Z 530.636,A -85,B 0,C 180,E1 -18794.076,E2 -18794.076} C_VEL
LIN {X 0,Y 248.324,Z 537.157,A -85,B 0,C 180,E1 -18796.914,E2 -18796.914} C_VEL
LIN {X 0,Y 247.398,Z 542.881,A -85,B 0,C 180,E1 -18800.187,E2 -18800.187} C_VEL
LIN {X 0,Y 247.152,Z 545.108,A -85,B 0,C 180,E1 -18801.826,E2 -18801.826} C_VEL
LIN {X 0,Y 246.845,Z 548.339,A -85,B 0,C 180,E1 -18805.1,E2 -18805.1} C_VEL
LIN {X 0,Y 246.922,Z 550.096,A -85,B 0,C 180,E1 -18808.369,E2 -18808.369} C_VEL
LIN {X 0,Y 246.982,Z 550.433,A -85,B 0,C 180,E1 -18810,E2 -18810} C_VEL
LIN {X 0,Y 246.923,Z 550.406,A -85,B 0,C 180,E1 -18811.631,E2 -18811.631} C_VEL
LIN {X 0,Y 246.881,Z 549.28,A -85,B 0,C 180,E1 -18814.899,E2 -18814.899} C_VEL
LIN {X 0,Y 247.158,Z 546.706,A -85,B 0,C 180,E1 -18818.174,E2 -18818.174} C_VEL
LIN {X 0,Y 247.865,Z 542.563,A -85,B 0,C 180,E1 -18821.448,E2 -18821.448} C_VEL
LIN {X 0,Y 248.84,Z 538.418,A -85,B 0,C 180,E1 -18823.89,E2 -18823.89} C_VEL
LIN {X 0,Y 250.14,Z 533.216,A -85,B 0,C 180,E1 -18826.317,E2 -18826.317} C_VEL
LIN {X 0,Y 252.065,Z 525.728,A -85,B 0,C 180,E1 -18829.123,E2 -18829.123} C_VEL
LIN {X 0,Y 254.146,Z 517.821,A -85,B 0,C 180,E1 -18831.494,E2 -18831.494} C_VEL
LIN {X 0,Y 256.689,Z 508.214,A -85,B 0,C 180,E1 -18833.818,E2 -18833.818} C_VEL
LIN {X 0,Y 259.484,Z 497.501,A -85,B 0,C 180,E1 -18835.896,E2 -18835.896} C_VEL
LIN {X 0,Y 261.968,Z 486.407,A -85,B 0,C 180,E1 -18837.643,E2 -18837.643} C_VEL
LIN {X 0,Y 264.525,Z 473.775,A -85,B 0,C 180,E1 -18839.221,E2 -18839.221} C_VEL
LIN {X 0,Y 266.766,Z 460.711,A -85,B 0,C 180,E1 -18840.473,E2 -18840.473} C_VEL
LIN {X 0,Y 268.697,Z 447.014,A -85,B 0,C 180,E1 -18841.431,E2 -18841.431} C_VEL
LIN {X 0,Y 270.085,Z 432.654,A -85,B 0,C 180,E1 -18842.127,E2 -18842.127} C_VEL
LIN {X 0,Y 271.308,Z 409.332,A -85,B 0,C 180,E1 -18842.789,E2 -18842.789} C_VEL
LIN {X 0,Y 273.995,Z 340.524,A -85,B 0,C 180,E1 -18844.63,E2 -18844.63} C_VEL
LIN {X 0,Y 273.154,Z 335.072,A -85,B 0,C 180,E1 -18844.927,E2 -18844.927} C_VEL
LIN {X 0,Y 266.423,Z 320.302,A -85,B 0,C 180,E1 -18846.43,E2 -18846.43} C_VEL
LIN {X 0,Y 260.333,Z 308.483,A -85,B 0,C 180,E1 -18847.824,E2 -18847.824} C_VEL
LIN {X 0,Y 256.576,Z 301.419,A -85,B 0,C 180,E1 -18848.784,E2 -18848.784} C_VEL
LIN {X 0,Y 254.139,Z 292.666,A -85,B 0,C 180,E1 -18852.29,E2 -18852.29} C_VEL
LIN {X 0,Y 251.631,Z 284.981,A -85,B 0,C 180,E1 -18855.714,E2 -18855.714} C_VEL
LIN {X 0,Y 249.026,Z 277.14,A -85,B 0,C 180,E1 -18859.639,E2 -18859.639} C_VEL
LIN {X 0,Y 249.028,Z 277.059,A -85,B 0,C 180,E1 -18863.655,E2 -18863.655} C_VEL
LIN {X 0,Y 249.034,Z 277.076,A -85,B 0,C 180,E1 -18867.846,E2 -18867.846} C_VEL
LIN {X 0,Y 249.083,Z 277.05,A -85,B 0,C 180,E1 -18871.337,E2 -18871.337} C_VEL
LIN {X 0,Y 249.148,Z 277.067,A -85,B 0,C 180,E1 -18874.969,E2 -18874.969} C_VEL
LIN {X 0,Y 249.107,Z 277.071,A -85,B 0,C 180,E1 -18880.212,E2 -18880.212} C_VEL
LIN {X 0,Y 249.239,Z 277.051,A -85,B 0,C 180,E1 -18883.622,E2 -18883.622} C_VEL
LIN {X 0,Y 249.249,Z 277.049,A -85,B 0,C 180,E1 -18888.617,E2 -18888.617} C_VEL
LIN {X 0,Y 249.476,Z 277.022,A -85,B 0,C 180,E1 -18891.903,E2 -18891.903} C_VEL
LIN {X 0,Y 249.432,Z 277.028,A -85,B 0,C 180,E1 -18896.77,E2 -18896.77} C_VEL
LIN {X 0,Y 249.724,Z 277.004,A -85,B 0,C 180,E1 -18900.001,E2 -18900.001} C_VEL
LIN {X 0,Y 249.433,Z 277.029,A -85,B 0,C 180,E1 -18903.231,E2 -18903.231} C_VEL
LIN {X 0,Y 249.478,Z 277.025,A -85,B 0,C 180,E1 -18908.098,E2 -18908.098} C_VEL
LIN {X 0,Y 249.25,Z 277.049,A -85,B 0,C 180,E1 -18911.384,E2 -18911.384} C_VEL
LIN {X 0,Y 249.216,Z 277.056,A -85,B 0,C 180,E1 -18916.504,E2 -18916.504} C_VEL
LIN {X 0,Y 249.086,Z 277.082,A -85,B 0,C 180,E1 -18921.519,E2 -18921.519} C_VEL
LIN {X 0,Y 249.129,Z 277.08,A -85,B 0,C 180,E1 -18925.483,E2 -18925.483} C_VEL
LIN {X 0,Y 249.072,Z 277.048,A -85,B 0,C 180,E1 -18928.99,E2 -18928.99} C_VEL
LIN {X 0,Y 249.035,Z 277.091,A -85,B 0,C 180,E1 -18932.426,E2 -18932.426} C_VEL
LIN {X 0,Y 249.069,Z 277.064,A -85,B 0,C 180,E1 -18936.34,E2 -18936.34} C_VEL
LIN {X 0,Y 249.076,Z 277.251,A -85,B 0,C 180,E1 -18938.372,E2 -18938.372} C_VEL
LIN {X 0,Y 251.417,Z 284.614,A -85,B 0,C 180,E1 -18942.136,E2 -18942.136} C_VEL
LIN {X 0,Y 253.992,Z 292.958,A -85,B 0,C 180,E1 -18946.008,E2 -18946.008} C_VEL
LIN {X 0,Y 256.29,Z 301.574,A -85,B 0,C 180,E1 -18949.619,E2 -18949.619} C_VEL
LIN {X 0,Y 258.315,Z 309.564,A -85,B 0,C 180,E1 -18952.624,E2 -18952.624} C_VEL
LIN {X 0,Y 266.192,Z 325.954,A -85,B 0,C 180,E1 -18954.476,E2 -18954.476} C_VEL
LIN {X 0,Y 267.676,Z 329.287,A -85,B 0,C 180,E1 -18954.808,E2 -18954.808} C_VEL
LIN {X 0,Y 272.222,Z 355.921,A -85,B 0,C 180,E1 -18956.285,E2 -18956.285} C_VEL
LIN {X 0,Y 272.958,Z 361.33,A -85,B 0,C 180,E1 -18956.55,E2 -18956.55} C_VEL
LIN {X 0,Y 270.441,Z 427.254,A -85,B 0,C 180,E1 -18958.185,E2 -18958.185} C_VEL
LIN {X 0,Y 269.17,Z 441.028,A -85,B 0,C 180,E1 -18958.794,E2 -18958.794} C_VEL
LIN {X 0,Y 267.499,Z 454.578,A -85,B 0,C 180,E1 -18959.728,E2 -18959.728} C_VEL
LIN {X 0,Y 265.531,Z 467.053,A -85,B 0,C 180,E1 -18960.925,E2 -18960.925} C_VEL
LIN {X 0,Y 263.247,Z 478.538,A -85,B 0,C 180,E1 -18962.364,E2 -18962.364} C_VEL
LIN {X 0,Y 260.675,Z 489.081,A -85,B 0,C 180,E1 -18964.017,E2 -18964.017} C_VEL
LIN {X 0,Y 258.081,Z 498.642,A -85,B 0,C 180,E1 -18965.891,E2 -18965.891} C_VEL
LIN {X 0,Y 255.366,Z 507.979,A -85,B 0,C 180,E1 -18968.19,E2 -18968.19} C_VEL
LIN {X 0,Y 253.088,Z 515.492,A -85,B 0,C 180,E1 -18970.535,E2 -18970.535} C_VEL
LIN {X 0,Y 251.31,Z 521.589,A -85,B 0,C 180,E1 -18972.924,E2 -18972.924} C_VEL
LIN {X 0,Y 249.74,Z 526.492,A -85,B 0,C 180,E1 -18975.329,E2 -18975.329} C_VEL
LIN {X 0,Y 248.598,Z 530.341,A -85,B 0,C 180,E1 -18977.759,E2 -18977.759} C_VEL
LIN {X 0,Y 247.836,Z 533.206,A -85,B 0,C 180,E1 -18980.204,E2 -18980.204} C_VEL
LIN {X 0,Y 247.438,Z 534.629,A -85,B 0,C 180,E1 -18981.836,E2 -18981.836} C_VEL
LIN {X 0,Y 247.014,Z 536.308,A -85,B 0,C 180,E1 -18985.104,E2 -18985.104} C_VEL
LIN {X 0,Y 246.983,Z 536.561,A -85,B 0,C 180,E1 -18988.369,E2 -18988.369} C_VEL
LIN {X 0,Y 247.086,Z 535.382,A -85,B 0,C 180,E1 -18991.63,E2 -18991.63} C_VEL
LIN {X 0,Y 247.605,Z 532.68,A -85,B 0,C 180,E1 -18994.885,E2 -18994.885} C_VEL
LIN {X 0,Y 248.481,Z 528.437,A -85,B 0,C 180,E1 -18998.13,E2 -18998.13} C_VEL
LIN {X 0,Y 249.455,Z 524.071,A -85,B 0,C 180,E1 -19000.552,E2 -19000.552} C_VEL
LIN {X 0,Y 251.116,Z 517.573,A -85,B 0,C 180,E1 -19003.349,E2 -19003.349} C_VEL
LIN {X 0,Y 252.999,Z 510.549,A -85,B 0,C 180,E1 -19005.714,E2 -19005.714} C_VEL
LIN {X 0,Y 255.168,Z 501.893,A -85,B 0,C 180,E1 -19008.05,E2 -19008.05} C_VEL
LIN {X 0,Y 257.212,Z 493.102,A -85,B 0,C 180,E1 -19009.971,E2 -19009.971} C_VEL
LIN {X 0,Y 259.631,Z 482.352,A -85,B 0,C 180,E1 -19011.851,E2 -19011.851} C_VEL
LIN {X 0,Y 261.744,Z 471.679,A -85,B 0,C 180,E1 -19013.331,E2 -19013.331} C_VEL
LIN {X 0,Y 263.723,Z 459.872,A -85,B 0,C 180,E1 -19014.606,E2 -19014.606} C_VEL
LIN {X 0,Y 265.217,Z 447.966,A -85,B 0,C 180,E1 -19015.594,E2 -19015.594} C_VEL
LIN {X 0,Y 266.462,Z 434.82,A -85,B 0,C 180,E1 -19016.366,E2 -19016.366} C_VEL
LIN {X 0,Y 267.263,Z 421.913,A -85,B 0,C 180,E1 -19016.834,E2 -19016.834} C_VEL
LIN {X 0,Y 269.345,Z 358.167,A -85,B 0,C 180,E1 -19018.422,E2 -19018.422} C_VEL
LIN {X 0,Y 264.967,Z 329.914,A -85,B 0,C 180,E1 -19019.832,E2 -19019.832} C_VEL
LIN {X 0,Y 263.462,Z 322.55,A -85,B 0,C 180,E1 -19020.26,E2 -19020.26} C_VEL
LIN {X 0,Y 257.674,Z 309.627,A -85,B 0,C 180,E1 -19021.545,E2 -19021.545} C_VEL
LIN {X 0,Y 255.561,Z 300.215,A -85,B 0,C 180,E1 -19024.902,E2 -19024.902} C_VEL
LIN {X 0,Y 253.311,Z 291.223,A -85,B 0,C 180,E1 -19028.456,E2 -19028.456} C_VEL
LIN {X 0,Y 250.64,Z 282.368,A -85,B 0,C 180,E1 -19032.295,E2 -19032.295} C_VEL
LIN {X 0,Y 249.006,Z 277.181,A -85,B 0,C 180,E1 -19034.77,E2 -19034.77} C_VEL
LIN {X 0,Y 249.009,Z 277.093,A -85,B 0,C 180,E1 -19037.36,E2 -19037.36} C_VEL
LIN {X 0,Y 249.037,Z 277.07,A -85,B 0,C 180,E1 -19041.621,E2 -19041.621} C_VEL
LIN {X 0,Y 249.06,Z 277.051,A -85,B 0,C 180,E1 -19045.641,E2 -19045.641} C_VEL
LIN {X 0,Y 249.049,Z 277.088,A -85,B 0,C 180,E1 -19049.472,E2 -19049.472} C_VEL
LIN {X 0,Y 249.072,Z 277.082,A -85,B 0,C 180,E1 -19053.161,E2 -19053.161} C_VEL
LIN {X 0,Y 249.077,Z 277.075,A -85,B 0,C 180,E1 -19056.732,E2 -19056.732} C_VEL
LIN {X 0,Y 249.107,Z 277.067,A -85,B 0,C 180,E1 -19060.211,E2 -19060.211} C_VEL
LIN {X 0,Y 249.239,Z 277.06,A -85,B 0,C 180,E1 -19063.621,E2 -19063.621} C_VEL
